  [744] = {x=191.932, y=87.653, z=110, rx=-180, rz=-113.182, shoulder=lefty, elbow=epositive, wrist=wpositive, fatherId=fReference[0]}
  [745] = {x=195.886, y=78.421, z=110, rx=-180, rz=-110.455, shoulder=lefty, elbow=epositive, wrist=wpositive, fatherId=fReference[0]}
  [746] = {x=199.395, y=69.011, z=110, rx=-180, rz=-107.727, shoulder=lefty, elbow=epositive, wrist=wpositive, fatherId=fReference[0]}
  [747] = {x=202.453, y=59.446, z=110, rx=-180, rz=-105, shoulder=lefty, elbow=epositive, wrist=wpositive, fatherId=fReference[0]}
  [748] = {x=205.052, y=49.745, z=110, rx=-180, rz=-102.273, shoulder=lefty, elbow=epositive, wrist=wpositive, fatherId=fReference[0]}
  [749] = {x=207.187, y=39.932, z=110, rx=-180, rz=-99.545, shoulder=lefty, elbow=epositive, wrist=wpositive, fatherId=fReference[0]}
  [750] = {x=208.852, y=30.028, z=110, rx=-180, rz=-96.818, shoulder=lefty, elbow=epositive, wrist=wpositive, fatherId=fReference[0]}
  [751] = {x=210.045, y=20.057, z=110, rx=-180, rz=-94.091, shoulder=lefty, elbow=epositive, wrist=wpositive, fatherId=fReference[0]}
  [752] = {x=210.761, y=10.04, z=110, rx=-180, rz=-91.364, shoulder=lefty, elbow=epositive, wrist=wpositive, fatherId=fReference[0]}
  [753] = {x=211, z=110, rx=180, rz=-88.636, shoulder=lefty, elbow=epositive, wrist=wpositive, fatherId=fReference[0]}
  [754] = {x=210.761, y=-10.04, z=110, rx=180, rz=-85.909, shoulder=lefty, elbow=epositive, wrist=wpositive, fatherId=fReference[0]}
  [755] = {x=210.045, y=-20.057, z=110, rx=180, rz=-83.182, shoulder=lefty, elbow=epositive, wrist=wpositive, fatherId=fReference[0]}
  [756] = {x=208.852, y=-30.028, z=110, rx=180, rz=-80.455, shoulder=lefty, elbow=epositive, wrist=wpositive, fatherId=fReference[0]}
  [757] = {x=207.187, y=-39.932, z=110, rx=180, rz=-77.727, shoulder=lefty, elbow=epositive, wrist=wpositive, fatherId=fReference[0]}
  [758] = {x=205.052, y=-49.745, z=110, rx=180, rz=-75, shoulder=lefty, elbow=epositive, wrist=wpositive, fatherId=fReference[0]}
  [759] = {x=202.453, y=-59.446, z=110, rx=180, rz=-72.273, shoulder=lefty, elbow=epositive, wrist=wpositive, fatherId=fReference[0]}
  [760] = {x=199.395, y=-69.011, z=110, rx=180, rz=-69.545, shoulder=lefty, elbow=epositive, wrist=wpositive, fatherId=fReference[0]}
  [761] = {x=195.886, y=-78.421, z=110, rx=180, rz=-66.818, shoulder=lefty, elbow=epositive, wrist=wpositive, fatherId=fReference[0]}
  [762] = {x=191.932, y=-87.653, z=110, rx=180, rz=-64.091, shoulder=lefty, elbow=epositive, wrist=wpositive, fatherId=fReference[0]}
  [763] = {x=187.544, y=-96.686, z=110, rx=180, rz=-61.364, shoulder=lefty, elbow=epositive, wrist=wpositive, fatherId=fReference[0]}
  [764] = {x=182.731, y=-105.5, z=110, rx=-180, rz=-58.636, shoulder=lefty, elbow=epositive, wrist=wpositive, fatherId=fReference[0]}
  [765] = {x=177.505, y=-114.075, z=110, rx=180, rz=-55.909, shoulder=lefty, elbow=epositive, wrist=wpositive, fatherId=fReference[0]}
  [766] = {x=171.876, y=-122.392, z=110, rx=180, rz=-53.182, shoulder=lefty, elbow=epositive, wrist=wpositive, fatherId=fReference[0]}
  [767] = {x=165.857, y=-130.432, z=110, rx=180, rz=-50.455, shoulder=lefty, elbow=epositive, wrist=wpositive, fatherId=fReference[0]}
  [768] = {x=159.463, y=-138.176, z=110, rx=180, rz=-47.727, shoulder=lefty, elbow=epositive, wrist=wpositive, fatherId=fReference[0]}
  [769] = {x=152.708, y=-145.607, z=110, rx=180, rz=-45, shoulder=lefty, elbow=epositive, wrist=wpositive, fatherId=fReference[0]}
  [770] = {x=145.607, y=-152.708, z=110, rx=180, rz=-42.273, shoulder=lefty, elbow=epositive, wrist=wpositive, fatherId=fReference[0]}
  [771] = {x=138.176, y=-159.463, z=110, rx=180, rz=-39.545, shoulder=lefty, elbow=epositive, wrist=wpositive, fatherId=fReference[0]}
  [772] = {x=130.432, y=-165.857, z=110, rx=-180, rz=-36.818, shoulder=lefty, elbow=epositive, wrist=wpositive, fatherId=fReference[0]}
  [773] = {x=122.392, y=-171.876, z=110, rx=180, rz=-34.091, shoulder=lefty, elbow=epositive, wrist=wpositive, fatherId=fReference[0]}
  [774] = {x=114.075, y=-177.505, z=110, rx=180, rz=-31.364, shoulder=lefty, elbow=epositive, wrist=wpositive, fatherId=fReference[0]}
  [775] = {x=105.5, y=-182.731, z=110, rx=-180, rz=-28.636, shoulder=lefty, elbow=epositive, wrist=wpositive, fatherId=fReference[0]}
  [776] = {x=96.686, y=-187.544, z=110, rx=-180, rz=-25.909, shoulder=lefty, elbow=epositive, wrist=wpositive, fatherId=fReference[0]}
  [777] = {x=87.653, y=-191.932, z=110, rx=180, rz=-23.182, shoulder=lefty, elbow=epositive, wrist=wpositive, fatherId=fReference[0]}
  [778] = {x=78.421, y=-195.886, z=110, rx=180, rz=-20.455, shoulder=lefty, elbow=epositive, wrist=wpositive, fatherId=fReference[0]}
  [779] = {x=69.011, y=-199.395, z=110, rx=-180, rz=-17.727, shoulder=lefty, elbow=epositive, wrist=wpositive, fatherId=fReference[0]}
  [780] = {x=59.446, y=-202.453, z=110, rx=180, rz=-15, shoulder=lefty, elbow=epositive, wrist=wpositive, fatherId=fReference[0]}
  [781] = {x=49.745, y=-205.052, z=110, rx=-180, rz=-12.273, shoulder=lefty, elbow=epositive, wrist=wpositive, fatherId=fReference[0]}
  [782] = {x=39.932, y=-207.187, z=110, rx=180, rz=-9.545, shoulder=lefty, elbow=epositive, wrist=wpositive, fatherId=fReference[0]}
  [783] = {x=30.028, y=-208.852, z=110, rx=-180, rz=-6.818, shoulder=lefty, elbow=epositive, wrist=wpositive, fatherId=fReference[0]}
  [784] = {x=20.057, y=-210.045, z=110, rx=180, rz=-4.091, shoulder=lefty, elbow=epositive, wrist=wpositive, fatherId=fReference[0]}
  [785] = {x=10.04, y=-210.761, z=110, rx=180, rz=-1.364, shoulder=lefty, elbow=epositive, wrist=wpositive, fatherId=fReference[0]}
  [786] = {y=-211, z=110, rx=-180, rz=1.364, shoulder=lefty, elbow=epositive, wrist=wpositive, fatherId=fReference[0]}
  [787] = {x=-10.04, y=-210.761, z=110, rx=-180, rz=4.091, shoulder=lefty, elbow=epositive, wrist=wpositive, fatherId=fReference[0]}
  [788] = {x=-20.057, y=-210.045, z=110, rx=-180, rz=6.818, shoulder=lefty, elbow=epositive, wrist=wpositive, fatherId=fReference[0]}
  [789] = {x=-30.028, y=-208.852, z=110, rx=-180, rz=9.545, shoulder=lefty, elbow=epositive, wrist=wpositive, fatherId=fReference[0]}
  [790] = {x=-39.932, y=-207.187, z=110, rx=-180, rz=12.273, shoulder=lefty, elbow=epositive, wrist=wpositive, fatherId=fReference[0]}
  [791] = {x=-49.745, y=-205.052, z=110, rx=-180, rz=15, shoulder=lefty, elbow=epositive, wrist=wpositive, fatherId=fReference[0]}
  [792] = {x=-59.446, y=-202.453, z=110, rx=-180, rz=17.727, shoulder=lefty, elbow=epositive, wrist=wpositive, fatherId=fReference[0]}
  [793] = {x=-69.011, y=-199.395, z=110, rx=-180, rz=20.455, shoulder=lefty, elbow=epositive, wrist=wpositive, fatherId=fReference[0]}
  [794] = {x=-78.421, y=-195.886, z=110, rx=-180, rz=23.182, shoulder=lefty, elbow=epositive, wrist=wpositive, fatherId=fReference[0]}
  [795] = {x=-87.653, y=-191.932, z=110, rx=-180, rz=25.909, shoulder=lefty, elbow=epositive, wrist=wpositive, fatherId=fReference[0]}
  [796] = {x=-96.686, y=-187.544, z=110, rx=-180, rz=28.636, shoulder=lefty, elbow=epositive, wrist=wpositive, fatherId=fReference[0]}
  [797] = {x=-105.5, y=-182.731, z=110, rx=-180, rz=31.364, shoulder=lefty, elbow=epositive, wrist=wpositive, fatherId=fReference[0]}
  [798] = {x=-114.075, y=-177.505, z=110, rx=-180, rz=34.091, shoulder=lefty, elbow=epositive, wrist=wpositive, fatherId=fReference[0]}
  [799] = {x=-122.392, y=-171.876, z=110, rx=-180, rz=36.818, shoulder=lefty, elbow=epositive, wrist=wpositive, fatherId=fReference[0]}
  [800] = {x=-130.432, y=-165.857, z=110, rx=-180, rz=39.545, shoulder=lefty, elbow=epositive, wrist=wpositive, fatherId=fReference[0]}
  [801] = {x=-138.176, y=-159.463, z=110, rx=-180, rz=42.273, shoulder=lefty, elbow=epositive, wrist=wpositive, fatherId=fReference[0]}
  [802] = {x=-145.607, y=-152.708, z=110, rx=-180, rz=45, shoulder=lefty, elbow=epositive, wrist=wpositive, fatherId=fReference[0]}
  [803] = {x=-152.708, y=-145.607, z=110, rx=-180, rz=47.727, shoulder=lefty, elbow=epositive, wrist=wpositive, fatherId=fReference[0]}
  [804] = {x=-159.463, y=-138.176, z=110, rx=180, rz=50.455, shoulder=lefty, elbow=epositive, wrist=wpositive, fatherId=fReference[0]}
  [805] = {x=-165.857, y=-130.432, z=110, rx=-180, rz=53.182, shoulder=lefty, elbow=epositive, wrist=wpositive, fatherId=fReference[0]}
  [806] = {x=-171.876, y=-122.392, z=110, rx=-180, rz=55.909, shoulder=lefty, elbow=epositive, wrist=wpositive, fatherId=fReference[0]}
  [807] = {x=-177.505, y=-114.075, z=110, rx=-180, rz=58.636, shoulder=lefty, elbow=epositive, wrist=wpositive, fatherId=fReference[0]}
  [808] = {x=-182.731, y=-105.5, z=110, rx=-180, rz=61.364, shoulder=lefty, elbow=epositive, wrist=wpositive, fatherId=fReference[0]}
  [809] = {x=-187.544, y=-96.686, z=110, rx=-180, rz=64.091, shoulder=lefty, elbow=epositive, wrist=wpositive, fatherId=fReference[0]}
  [810] = {x=-191.932, y=-87.653, z=110, rx=180, rz=66.818, shoulder=lefty, elbow=epositive, wrist=wpositive, fatherId=fReference[0]}
  [811] = {x=-195.886, y=-78.421, z=110, rx=-180, rz=69.545, shoulder=lefty, elbow=epositive, wrist=wpositive, fatherId=fReference[0]}
  [812] = {x=-199.395, y=-69.011, z=110, rx=-180, rz=72.273, shoulder=lefty, elbow=epositive, wrist=wpositive, fatherId=fReference[0]}
  [813] = {x=-202.453, y=-59.446, z=110, rx=-180, rz=75, shoulder=lefty, elbow=epositive, wrist=wpositive, fatherId=fReference[0]}
  [814] = {x=-205.052, y=-49.745, z=110, rx=-180, rz=77.727, shoulder=lefty, elbow=epositive, wrist=wpositive, fatherId=fReference[0]}
  [815] = {x=-207.187, y=-39.932, z=110, rx=-180, rz=80.455, shoulder=lefty, elbow=epositive, wrist=wpositive, fatherId=fReference[0]}
  [816] = {x=-208.852, y=-30.028, z=110, rx=-180, rz=83.182, shoulder=lefty, elbow=epositive, wrist=wpositive, fatherId=fReference[0]}
  [817] = {x=-210.045, y=-20.057, z=110, rx=-180, rz=85.909, shoulder=lefty, elbow=epositive, wrist=wpositive, fatherId=fReference[0]}
  [818] = {x=-210.761, y=-10.04, z=110, rx=-180, rz=88.636, shoulder=lefty, elbow=epositive, wrist=wpositive, fatherId=fReference[0]}
  [819] = {x=-211, z=110, rx=-180, rz=88.636, shoulder=lefty, elbow=epositive, wrist=wpositive, fatherId=fReference[0]}
  [820] = {x=-211, z=110, rx=-180, rz=88.636, shoulder=lefty, elbow=epositive, wrist=wpositive, fatherId=fReference[0]}
  [821] = {x=-211, z=210, rx=-180, rz=88.636, shoulder=lefty, elbow=epositive, wrist=wpositive, fatherId=fReference[0]}
  [822] = {x=-211, z=232, rx=-180, rz=88.636, shoulder=lefty, elbow=epositive, wrist=wpositive, fatherId=fReference[0]}
  [823] = {x=-211, z=132, rx=-180, rz=88.636, shoulder=lefty, elbow=epositive, wrist=wpositive, fatherId=fReference[0]}
  [824] = {x=-211, z=132, rx=-180, rz=88.636, shoulder=lefty, elbow=epositive, wrist=wpositive, fatherId=fReference[0]}
  [825] = {x=-210.761, y=-10.04, z=132, rx=-180, rz=85.909, shoulder=lefty, elbow=epositive, wrist=wpositive, fatherId=fReference[0]}
  [826] = {x=-210.045, y=-20.057, z=132, rx=-180, rz=83.182, shoulder=lefty, elbow=epositive, wrist=wpositive, fatherId=fReference[0]}
  [827] = {x=-208.852, y=-30.028, z=132, rx=-180, rz=80.455, shoulder=lefty, elbow=epositive, wrist=wpositive, fatherId=fReference[0]}
  [828] = {x=-207.187, y=-39.932, z=132, rx=-180, rz=77.727, shoulder=lefty, elbow=epositive, wrist=wpositive, fatherId=fReference[0]}
  [829] = {x=-205.052, y=-49.745, z=132, rx=-180, rz=75, shoulder=lefty, elbow=epositive, wrist=wpositive, fatherId=fReference[0]}
  [830] = {x=-202.453, y=-59.446, z=132, rx=-180, rz=72.273, shoulder=lefty, elbow=epositive, wrist=wpositive, fatherId=fReference[0]}
  [831] = {x=-199.395, y=-69.011, z=132, rx=-180, rz=69.545, shoulder=lefty, elbow=epositive, wrist=wpositive, fatherId=fReference[0]}
  [832] = {x=-195.886, y=-78.421, z=132, rx=-180, rz=66.818, shoulder=lefty, elbow=epositive, wrist=wpositive, fatherId=fReference[0]}
  [833] = {x=-191.932, y=-87.653, z=132, rx=180, rz=64.091, shoulder=lefty, elbow=epositive, wrist=wpositive, fatherId=fReference[0]}
  [834] = {x=-187.544, y=-96.686, z=132, rx=-180, rz=61.364, shoulder=lefty, elbow=epositive, wrist=wpositive, fatherId=fReference[0]}
  [835] = {x=-182.731, y=-105.5, z=132, rx=-180, rz=58.636, shoulder=lefty, elbow=epositive, wrist=wpositive, fatherId=fReference[0]}
  [836] = {x=-177.505, y=-114.075, z=132, rx=180, rz=55.909, shoulder=lefty, elbow=epositive, wrist=wpositive, fatherId=fReference[0]}
  [837] = {x=-171.876, y=-122.392, z=132, rx=-180, rz=53.182, shoulder=lefty, elbow=epositive, wrist=wpositive, fatherId=fReference[0]}
  [838] = {x=-165.857, y=-130.432, z=132, rx=-180, rz=50.455, shoulder=lefty, elbow=epositive, wrist=wpositive, fatherId=fReference[0]}
  [839] = {x=-159.463, y=-138.176, z=132, rx=-180, rz=47.727, shoulder=lefty, elbow=epositive, wrist=wpositive, fatherId=fReference[0]}
  [840] = {x=-152.708, y=-145.607, z=132, rx=-180, rz=45, shoulder=lefty, elbow=epositive, wrist=wpositive, fatherId=fReference[0]}
  [841] = {x=-145.607, y=-152.708, z=132, rx=-180, rz=42.273, shoulder=lefty, elbow=epositive, wrist=wpositive, fatherId=fReference[0]}
  [842] = {x=-138.176, y=-159.463, z=132, rx=180, rz=39.545, shoulder=lefty, elbow=epositive, wrist=wpositive, fatherId=fReference[0]}
  [843] = {x=-130.432, y=-165.857, z=132, rx=-180, rz=36.818, shoulder=lefty, elbow=epositive, wrist=wpositive, fatherId=fReference[0]}
  [844] = {x=-122.392, y=-171.876, z=132, rx=-180, rz=34.091, shoulder=lefty, elbow=epositive, wrist=wpositive, fatherId=fReference[0]}
  [845] = {x=-114.075, y=-177.505, z=132, rx=-180, rz=31.364, shoulder=lefty, elbow=epositive, wrist=wpositive, fatherId=fReference[0]}
  [846] = {x=-105.5, y=-182.731, z=132, rx=180, rz=28.636, shoulder=lefty, elbow=epositive, wrist=wpositive, fatherId=fReference[0]}
  [847] = {x=-96.686, y=-187.544, z=132, rx=-180, rz=25.909, shoulder=lefty, elbow=epositive, wrist=wpositive, fatherId=fReference[0]}
  [848] = {x=-87.653, y=-191.932, z=132, rx=180, rz=23.182, shoulder=lefty, elbow=epositive, wrist=wpositive, fatherId=fReference[0]}
  [849] = {x=-78.421, y=-195.886, z=132, rx=180, rz=20.455, shoulder=lefty, elbow=epositive, wrist=wpositive, fatherId=fReference[0]}
  [850] = {x=-69.011, y=-199.395, z=132, rx=-180, rz=17.727, shoulder=lefty, elbow=epositive, wrist=wpositive, fatherId=fReference[0]}
  [851] = {x=-59.446, y=-202.453, z=132, rx=180, rz=15, shoulder=lefty, elbow=epositive, wrist=wpositive, fatherId=fReference[0]}
  [852] = {x=-49.745, y=-205.052, z=132, rx=-180, rz=12.273, shoulder=lefty, elbow=epositive, wrist=wpositive, fatherId=fReference[0]}
  [853] = {x=-39.932, y=-207.187, z=132, rx=180, rz=9.545, shoulder=lefty, elbow=epositive, wrist=wpositive, fatherId=fReference[0]}
  [854] = {x=-30.028, y=-208.852, z=132, rx=-180, rz=6.818, shoulder=lefty, elbow=epositive, wrist=wpositive, fatherId=fReference[0]}
  [855] = {x=-20.057, y=-210.045, z=132, rx=180, rz=4.091, shoulder=lefty, elbow=epositive, wrist=wpositive, fatherId=fReference[0]}
  [856] = {x=-10.04, y=-210.761, z=132, rx=-180, rz=1.364, shoulder=lefty, elbow=epositive, wrist=wpositive, fatherId=fReference[0]}
  [857] = {y=-211, z=132, rx=180, rz=-1.364, shoulder=lefty, elbow=epositive, wrist=wpositive, fatherId=fReference[0]}
  [858] = {x=10.04, y=-210.761, z=132, rx=180, rz=-4.091, shoulder=lefty, elbow=epositive, wrist=wpositive, fatherId=fReference[0]}
  [859] = {x=20.057, y=-210.045, z=132, rx=180, rz=-6.818, shoulder=lefty, elbow=epositive, wrist=wpositive, fatherId=fReference[0]}
  [860] = {x=30.028, y=-208.852, z=132, rx=180, rz=-9.545, shoulder=lefty, elbow=epositive, wrist=wpositive, fatherId=fReference[0]}
  [861] = {x=39.932, y=-207.187, z=132, rx=180, rz=-12.273, shoulder=lefty, elbow=epositive, wrist=wpositive, fatherId=fReference[0]}
  [862] = {x=49.745, y=-205.052, z=132, rx=-180, rz=-15, shoulder=lefty, elbow=epositive, wrist=wpositive, fatherId=fReference[0]}
  [863] = {x=59.446, y=-202.453, z=132, rx=-180, rz=-17.727, shoulder=lefty, elbow=epositive, wrist=wpositive, fatherId=fReference[0]}
  [864] = {x=69.011, y=-199.395, z=132, rx=180, rz=-20.455, shoulder=lefty, elbow=epositive, wrist=wpositive, fatherId=fReference[0]}
  [865] = {x=78.421, y=-195.886, z=132, rx=-180, rz=-23.182, shoulder=lefty, elbow=epositive, wrist=wpositive, fatherId=fReference[0]}
  [866] = {x=87.653, y=-191.932, z=132, rx=-180, rz=-25.909, shoulder=lefty, elbow=epositive, wrist=wpositive, fatherId=fReference[0]}
  [867] = {x=96.686, y=-187.544, z=132, rx=-180, rz=-28.636, shoulder=lefty, elbow=epositive, wrist=wpositive, fatherId=fReference[0]}
  [868] = {x=105.5, y=-182.731, z=132, rx=180, rz=-31.364, shoulder=lefty, elbow=epositive, wrist=wpositive, fatherId=fReference[0]}
  [869] = {x=114.075, y=-177.505, z=132, rx=180, rz=-34.091, shoulder=lefty, elbow=epositive, wrist=wpositive, fatherId=fReference[0]}
  [870] = {x=122.392, y=-171.876, z=132, rx=180, rz=-36.818, shoulder=lefty, elbow=epositive, wrist=wpositive, fatherId=fReference[0]}
  [871] = {x=130.432, y=-165.857, z=132, rx=180, rz=-39.545, shoulder=lefty, elbow=epositive, wrist=wpositive, fatherId=fReference[0]}
  [872] = {x=138.176, y=-159.463, z=132, rx=180, rz=-42.273, shoulder=lefty, elbow=epositive, wrist=wpositive, fatherId=fReference[0]}
  [873] = {x=145.607, y=-152.708, z=132, rx=180, rz=-45, shoulder=lefty, elbow=epositive, wrist=wpositive, fatherId=fReference[0]}
  [874] = {x=152.708, y=-145.607, z=132, rx=180, rz=-47.727, shoulder=lefty, elbow=epositive, wrist=wpositive, fatherId=fReference[0]}
  [875] = {x=159.463, y=-138.176, z=132, rx=180, rz=-50.455, shoulder=lefty, elbow=epositive, wrist=wpositive, fatherId=fReference[0]}
  [876] = {x=165.857, y=-130.432, z=132, rx=180, rz=-53.182, shoulder=lefty, elbow=epositive, wrist=wpositive, fatherId=fReference[0]}
  [877] = {x=171.876, y=-122.392, z=132, rx=180, rz=-55.909, shoulder=lefty, elbow=epositive, wrist=wpositive, fatherId=fReference[0]}
  [878] = {x=177.505, y=-114.075, z=132, rx=180, rz=-58.636, shoulder=lefty, elbow=epositive, wrist=wpositive, fatherId=fReference[0]}
  [879] = {x=182.731, y=-105.5, z=132, rx=180, rz=-61.364, shoulder=lefty, elbow=epositive, wrist=wpositive, fatherId=fReference[0]}
  [880] = {x=187.544, y=-96.686, z=132, rx=180, rz=-64.091, shoulder=lefty, elbow=epositive, wrist=wpositive, fatherId=fReference[0]}
  [881] = {x=191.932, y=-87.653, z=132, rx=-180, rz=-66.818, shoulder=lefty, elbow=epositive, wrist=wpositive, fatherId=fReference[0]}
  [882] = {x=195.886, y=-78.421, z=132, rx=180, rz=-69.545, shoulder=lefty, elbow=epositive, wrist=wpositive, fatherId=fReference[0]}
  [883] = {x=199.395, y=-69.011, z=132, rx=180, rz=-72.273, shoulder=lefty, elbow=epositive, wrist=wpositive, fatherId=fReference[0]}
  [884] = {x=202.453, y=-59.446, z=132, rx=180, rz=-75, shoulder=lefty, elbow=epositive, wrist=wpositive, fatherId=fReference[0]}
  [885] = {x=205.052, y=-49.745, z=132, rx=180, rz=-77.727, shoulder=lefty, elbow=epositive, wrist=wpositive, fatherId=fReference[0]}
  [886] = {x=207.187, y=-39.932, z=132, rx=180, rz=-80.455, shoulder=lefty, elbow=epositive, wrist=wpositive, fatherId=fReference[0]}
  [887] = {x=208.852, y=-30.028, z=132, rx=180, rz=-83.182, shoulder=lefty, elbow=epositive, wrist=wpositive, fatherId=fReference[0]}
  [888] = {x=210.045, y=-20.057, z=132, rx=180, rz=-85.909, shoulder=lefty, elbow=epositive, wrist=wpositive, fatherId=fReference[0]}
  [889] = {x=210.761, y=-10.04, z=132, rx=180, rz=-88.636, shoulder=lefty, elbow=epositive, wrist=wpositive, fatherId=fReference[0]}
  [890] = {x=211, z=132, rx=-180, rz=-91.364, shoulder=lefty, elbow=epositive, wrist=wpositive, fatherId=fReference[0]}
  [891] = {x=210.761, y=10.04, z=132, rx=-180, rz=-94.091, shoulder=lefty, elbow=epositive, wrist=wpositive, fatherId=fReference[0]}
  [892] = {x=210.045, y=20.057, z=132, rx=-180, rz=-96.818, shoulder=lefty, elbow=epositive, wrist=wpositive, fatherId=fReference[0]}
  [893] = {x=208.852, y=30.028, z=132, rx=-180, rz=-99.545, shoulder=lefty, elbow=epositive, wrist=wpositive, fatherId=fReference[0]}
  [894] = {x=207.187, y=39.932, z=132, rx=-180, rz=-102.273, shoulder=lefty, elbow=epositive, wrist=wpositive, fatherId=fReference[0]}
  [895] = {x=205.052, y=49.745, z=132, rx=-180, rz=-105, shoulder=lefty, elbow=epositive, wrist=wpositive, fatherId=fReference[0]}
  [896] = {x=202.453, y=59.446, z=132, rx=-180, rz=-107.727, shoulder=lefty, elbow=epositive, wrist=wpositive, fatherId=fReference[0]}
  [897] = {x=199.395, y=69.011, z=132, rx=-180, rz=-110.455, shoulder=lefty, elbow=epositive, wrist=wpositive, fatherId=fReference[0]}
  [898] = {x=195.886, y=78.421, z=132, rx=-180, rz=-113.182, shoulder=lefty, elbow=epositive, wrist=wpositive, fatherId=fReference[0]}
  [899] = {x=191.932, y=87.653, z=132, rx=-180, rz=-115.909, shoulder=lefty, elbow=epositive, wrist=wpositive, fatherId=fReference[0]}
  [900] = {x=187.544, y=96.686, z=132, rx=-180, rz=-118.636, shoulder=lefty, elbow=epositive, wrist=wpositive, fatherId=fReference[0]}
  [901] = {x=182.731, y=105.5, z=132, rx=-180, rz=-121.364, shoulder=lefty, elbow=epositive, wrist=wpositive, fatherId=fReference[0]}
  [902] = {x=177.505, y=114.075, z=132, rx=-180, rz=-124.091, shoulder=lefty, elbow=epositive, wrist=wpositive, fatherId=fReference[0]}
  [903] = {x=171.876, y=122.392, z=132, rx=-180, rz=-126.818, shoulder=lefty, elbow=epositive, wrist=wpositive, fatherId=fReference[0]}
  [904] = {x=165.857, y=130.432, z=132, rx=-180, rz=-129.545, shoulder=lefty, elbow=epositive, wrist=wpositive, fatherId=fReference[0]}
  [905] = {x=159.463, y=138.176, z=132, rx=-180, rz=-132.273, shoulder=lefty, elbow=epositive, wrist=wpositive, fatherId=fReference[0]}
  [906] = {x=152.708, y=145.607, z=132, rx=-180, rz=-135, shoulder=lefty, elbow=epositive, wrist=wpositive, fatherId=fReference[0]}
  [907] = {x=145.607, y=152.708, z=132, rx=-180, rz=-137.727, shoulder=lefty, elbow=epositive, wrist=wpositive, fatherId=fReference[0]}
  [908] = {x=138.176, y=159.463, z=132, rx=-180, rz=-140.455, shoulder=lefty, elbow=epositive, wrist=wpositive, fatherId=fReference[0]}
  [909] = {x=130.432, y=165.857, z=132, rx=180, rz=-143.182, shoulder=lefty, elbow=epositive, wrist=wpositive, fatherId=fReference[0]}
  [910] = {x=122.392, y=171.876, z=132, rx=-180, rz=-145.909, shoulder=lefty, elbow=epositive, wrist=wpositive, fatherId=fReference[0]}
  [911] = {x=114.075, y=177.505, z=132, rx=180, rz=-148.636, shoulder=lefty, elbow=epositive, wrist=wpositive, fatherId=fReference[0]}
  [912] = {x=105.5, y=182.731, z=132, rx=180, rz=-151.364, shoulder=lefty, elbow=epositive, wrist=wpositive, fatherId=fReference[0]}
  [913] = {x=96.686, y=187.544, z=132, rx=-180, rz=-154.091, shoulder=lefty, elbow=epositive, wrist=wpositive, fatherId=fReference[0]}
  [914] = {x=87.653, y=191.932, z=132, rx=-180, rz=-156.818, shoulder=lefty, elbow=epositive, wrist=wpositive, fatherId=fReference[0]}
  [915] = {x=78.421, y=195.886, z=132, rx=-180, rz=-159.545, shoulder=lefty, elbow=epositive, wrist=wpositive, fatherId=fReference[0]}
  [916] = {x=69.011, y=199.395, z=132, rx=-180, rz=-162.273, shoulder=lefty, elbow=epositive, wrist=wpositive, fatherId=fReference[0]}
  [917] = {x=59.446, y=202.453, z=132, rx=-180, rz=-165, shoulder=lefty, elbow=epositive, wrist=wpositive, fatherId=fReference[0]}
  [918] = {x=49.745, y=205.052, z=132, rx=180, rz=-167.727, shoulder=lefty, elbow=epositive, wrist=wpositive, fatherId=fReference[0]}
  [919] = {x=39.932, y=207.187, z=132, rx=180, rz=-170.455, shoulder=lefty, elbow=epositive, wrist=wpositive, fatherId=fReference[0]}
  [920] = {x=30.028, y=208.852, z=132, rx=-180, rz=-173.182, shoulder=lefty, elbow=epositive, wrist=wpositive, fatherId=fReference[0]}
  [921] = {x=20.057, y=210.045, z=132, rx=-180, rz=-175.909, shoulder=lefty, elbow=epositive, wrist=wpositive, fatherId=fReference[0]}
  [922] = {x=10.04, y=210.761, z=132, rx=-180, rz=-178.636, shoulder=lefty, elbow=epositive, wrist=wpositive, fatherId=fReference[0]}
  [923] = {y=211, z=132, rx=-180, rz=178.636, shoulder=lefty, elbow=epositive, wrist=wpositive, fatherId=fReference[0]}
  [924] = {x=-10.04, y=210.761, z=132, rx=180, rz=175.909, shoulder=lefty, elbow=epositive, wrist=wpositive, fatherId=fReference[0]}
  [925] = {x=-20.057, y=210.045, z=132, rx=180, rz=173.182, shoulder=lefty, elbow=epositive, wrist=wpositive, fatherId=fReference[0]}
  [926] = {x=-30.028, y=208.852, z=132, rx=180, rz=170.455, shoulder=lefty, elbow=epositive, wrist=wpositive, fatherId=fReference[0]}
  [927] = {x=-39.932, y=207.187, z=132, rx=180, rz=167.727, shoulder=lefty, elbow=epositive, wrist=wpositive, fatherId=fReference[0]}
  [928] = {x=-49.745, y=205.052, z=132, rx=-180, rz=165, shoulder=lefty, elbow=epositive, wrist=wpositive, fatherId=fReference[0]}
  [929] = {x=-59.446, y=202.453, z=132, rx=180, rz=162.273, shoulder=lefty, elbow=epositive, wrist=wpositive, fatherId=fReference[0]}
  [930] = {x=-69.011, y=199.395, z=132, rx=180, rz=159.545, shoulder=lefty, elbow=epositive, wrist=wpositive, fatherId=fReference[0]}
  [931] = {x=-78.421, y=195.886, z=132, rx=-180, rz=156.818, shoulder=lefty, elbow=epositive, wrist=wpositive, fatherId=fReference[0]}
  [932] = {x=-87.653, y=191.932, z=132, rx=180, rz=154.091, shoulder=lefty, elbow=epositive, wrist=wpositive, fatherId=fReference[0]}
  [933] = {x=-96.686, y=187.544, z=132, rx=-180, rz=151.364, shoulder=lefty, elbow=epositive, wrist=wpositive, fatherId=fReference[0]}
  [934] = {x=-105.5, y=182.731, z=132, rx=180, rz=148.636, shoulder=lefty, elbow=epositive, wrist=wpositive, fatherId=fReference[0]}
  [935] = {x=-114.075, y=177.505, z=132, rx=-180, rz=145.909, shoulder=lefty, elbow=epositive, wrist=wpositive, fatherId=fReference[0]}
  [936] = {x=-122.392, y=171.876, z=132, rx=-180, rz=143.182, shoulder=lefty, elbow=epositive, wrist=wpositive, fatherId=fReference[0]}
  [937] = {x=-130.432, y=165.857, z=132, rx=-180, rz=140.455, shoulder=lefty, elbow=epositive, wrist=wpositive, fatherId=fReference[0]}
  [938] = {x=-138.176, y=159.463, z=132, rx=180, rz=137.727, shoulder=lefty, elbow=epositive, wrist=wpositive, fatherId=fReference[0]}
  [939] = {x=-145.607, y=152.708, z=132, rx=180, rz=135, shoulder=lefty, elbow=epositive, wrist=wpositive, fatherId=fReference[0]}
  [940] = {x=-152.708, y=145.607, z=132, rx=180, rz=132.273, shoulder=lefty, elbow=epositive, wrist=wpositive, fatherId=fReference[0]}
  [941] = {x=-159.463, y=138.176, z=132, rx=180, rz=129.545, shoulder=lefty, elbow=epositive, wrist=wpositive, fatherId=fReference[0]}
  [942] = {x=-165.857, y=130.432, z=132, rx=180, rz=126.818, shoulder=lefty, elbow=epositive, wrist=wpositive, fatherId=fReference[0]}
  [943] = {x=-171.876, y=122.392, z=132, rx=180, rz=124.091, shoulder=lefty, elbow=epositive, wrist=wpositive, fatherId=fReference[0]}
  [944] = {x=-177.505, y=114.075, z=132, rx=180, rz=121.364, shoulder=lefty, elbow=epositive, wrist=wpositive, fatherId=fReference[0]}
  [945] = {x=-182.731, y=105.5, z=132, rx=180, rz=118.636, shoulder=lefty, elbow=epositive, wrist=wpositive, fatherId=fReference[0]}
  [946] = {x=-187.544, y=96.686, z=132, rx=180, rz=115.909, shoulder=lefty, elbow=epositive, wrist=wpositive, fatherId=fReference[0]}
  [947] = {x=-191.932, y=87.653, z=132, rx=180, rz=113.182, shoulder=lefty, elbow=epositive, wrist=wpositive, fatherId=fReference[0]}
  [948] = {x=-195.886, y=78.421, z=132, rx=180, rz=110.455, shoulder=lefty, elbow=epositive, wrist=wpositive, fatherId=fReference[0]}
  [949] = {x=-199.395, y=69.011, z=132, rx=180, rz=107.727, shoulder=lefty, elbow=epositive, wrist=wpositive, fatherId=fReference[0]}
  [950] = {x=-202.453, y=59.446, z=132, rx=180, rz=105, shoulder=lefty, elbow=epositive, wrist=wpositive, fatherId=fReference[0]}
  [951] = {x=-205.052, y=49.745, z=132, rx=180, rz=102.273, shoulder=lefty, elbow=epositive, wrist=wpositive, fatherId=fReference[0]}
  [952] = {x=-207.187, y=39.932, z=132, rx=180, rz=99.545, shoulder=lefty, elbow=epositive, wrist=wpositive, fatherId=fReference[0]}
  [953] = {x=-208.852, y=30.028, z=132, rx=180, rz=96.818, shoulder=lefty, elbow=epositive, wrist=wpositive, fatherId=fReference[0]}
  [954] = {x=-210.045, y=20.057, z=132, rx=180, rz=94.091, shoulder=lefty, elbow=epositive, wrist=wpositive, fatherId=fReference[0]}
  [955] = {x=-210.761, y=10.04, z=132, rx=180, rz=91.364, shoulder=lefty, elbow=epositive, wrist=wpositive, fatherId=fReference[0]}
  [956] = {x=-211, z=132, rx=180, rz=91.364, shoulder=lefty, elbow=epositive, wrist=wpositive, fatherId=fReference[0]}
  [957] = {x=-211, z=132, rx=180, rz=91.364, shoulder=lefty, elbow=epositive, wrist=wpositive, fatherId=fReference[0]}
  [958] = {x=-211, z=232, rx=180, rz=91.364, shoulder=lefty, elbow=epositive, wrist=wpositive, fatherId=fReference[0]}
  [959] = {x=-211, z=254, rx=180, rz=91.364, shoulder=lefty, elbow=epositive, wrist=wpositive, fatherId=fReference[0]}
  [960] = {x=-211, z=154, rx=180, rz=91.364, shoulder=lefty, elbow=epositive, wrist=wpositive, fatherId=fReference[0]}
  [961] = {x=-211, z=154, rx=180, rz=91.364, shoulder=lefty, elbow=epositive, wrist=wpositive, fatherId=fReference[0]}
  [962] = {x=-210.761, y=10.04, z=154, rx=180, rz=94.091, shoulder=lefty, elbow=epositive, wrist=wpositive, fatherId=fReference[0]}
  [963] = {x=-210.045, y=20.057, z=154, rx=180, rz=96.818, shoulder=lefty, elbow=epositive, wrist=wpositive, fatherId=fReference[0]}
  [964] = {x=-208.852, y=30.028, z=154, rx=180, rz=99.545, shoulder=lefty, elbow=epositive, wrist=wpositive, fatherId=fReference[0]}
  [965] = {x=-207.187, y=39.932, z=154, rx=180, rz=102.273, shoulder=lefty, elbow=epositive, wrist=wpositive, fatherId=fReference[0]}
  [966] = {x=-205.052, y=49.745, z=154, rx=180, rz=105, shoulder=lefty, elbow=epositive, wrist=wpositive, fatherId=fReference[0]}
  [967] = {x=-202.453, y=59.446, z=154, rx=180, rz=107.727, shoulder=lefty, elbow=epositive, wrist=wpositive, fatherId=fReference[0]}
  [968] = {x=-199.395, y=69.011, z=154, rx=180, rz=110.455, shoulder=lefty, elbow=epositive, wrist=wpositive, fatherId=fReference[0]}
  [969] = {x=-195.886, y=78.421, z=154, rx=180, rz=113.182, shoulder=lefty, elbow=epositive, wrist=wpositive, fatherId=fReference[0]}
  [970] = {x=-191.932, y=87.653, z=154, rx=180, rz=115.909, shoulder=lefty, elbow=epositive, wrist=wpositive, fatherId=fReference[0]}
  [971] = {x=-187.544, y=96.686, z=154, rx=180, rz=118.636, shoulder=lefty, elbow=epositive, wrist=wpositive, fatherId=fReference[0]}
  [972] = {x=-182.731, y=105.5, z=154, rx=180, rz=121.364, shoulder=lefty, elbow=epositive, wrist=wpositive, fatherId=fReference[0]}
  [973] = {x=-177.505, y=114.075, z=154, rx=180, rz=124.091, shoulder=lefty, elbow=epositive, wrist=wpositive, fatherId=fReference[0]}
  [974] = {x=-171.876, y=122.392, z=154, rx=180, rz=126.818, shoulder=lefty, elbow=epositive, wrist=wpositive, fatherId=fReference[0]}
  [975] = {x=-165.857, y=130.432, z=154, rx=180, rz=129.545, shoulder=lefty, elbow=epositive, wrist=wpositive, fatherId=fReference[0]}
  [976] = {x=-159.463, y=138.176, z=154, rx=180, rz=132.273, shoulder=lefty, elbow=epositive, wrist=wpositive, fatherId=fReference[0]}
  [977] = {x=-152.708, y=145.607, z=154, rx=-180, rz=135, shoulder=lefty, elbow=epositive, wrist=wpositive, fatherId=fReference[0]}
  [978] = {x=-145.607, y=152.708, z=154, rx=-180, rz=137.727, shoulder=lefty, elbow=epositive, wrist=wpositive, fatherId=fReference[0]}
  [979] = {x=-138.176, y=159.463, z=154, rx=180, rz=140.455, shoulder=lefty, elbow=epositive, wrist=wpositive, fatherId=fReference[0]}
  [980] = {x=-130.432, y=165.857, z=154, rx=180, rz=143.182, shoulder=lefty, elbow=epositive, wrist=wpositive, fatherId=fReference[0]}
  [981] = {x=-122.392, y=171.876, z=154, rx=180, rz=145.909, shoulder=lefty, elbow=epositive, wrist=wpositive, fatherId=fReference[0]}
  [982] = {x=-114.075, y=177.505, z=154, rx=180, rz=148.636, shoulder=lefty, elbow=epositive, wrist=wpositive, fatherId=fReference[0]}
  [983] = {x=-105.5, y=182.731, z=154, rx=180, rz=151.364, shoulder=lefty, elbow=epositive, wrist=wpositive, fatherId=fReference[0]}
  [984] = {x=-96.686, y=187.544, z=154, rx=-180, rz=154.091, shoulder=lefty, elbow=epositive, wrist=wpositive, fatherId=fReference[0]}
  [985] = {x=-87.653, y=191.932, z=154, rx=-180, rz=156.818, shoulder=lefty, elbow=epositive, wrist=wpositive, fatherId=fReference[0]}
  [986] = {x=-78.421, y=195.886, z=154, rx=180, rz=159.545, shoulder=lefty, elbow=epositive, wrist=wpositive, fatherId=fReference[0]}
  [987] = {x=-69.011, y=199.395, z=154, rx=-180, rz=162.273, shoulder=lefty, elbow=epositive, wrist=wpositive, fatherId=fReference[0]}
  [988] = {x=-59.446, y=202.453, z=154, rx=180, rz=165, shoulder=lefty, elbow=epositive, wrist=wpositive, fatherId=fReference[0]}
  [989] = {x=-49.745, y=205.052, z=154, rx=180, rz=167.727, shoulder=lefty, elbow=epositive, wrist=wpositive, fatherId=fReference[0]}
  [990] = {x=-39.932, y=207.187, z=154, rx=180, rz=170.455, shoulder=lefty, elbow=epositive, wrist=wpositive, fatherId=fReference[0]}
  [991] = {x=-30.028, y=208.852, z=154, rx=-180, rz=173.182, shoulder=lefty, elbow=epositive, wrist=wpositive, fatherId=fReference[0]}
  [992] = {x=-20.057, y=210.045, z=154, rx=-180, rz=175.909, shoulder=lefty, elbow=epositive, wrist=wpositive, fatherId=fReference[0]}
  [993] = {x=-10.04, y=210.761, z=154, rx=-180, rz=178.636, shoulder=lefty, elbow=epositive, wrist=wpositive, fatherId=fReference[0]}
  [994] = {y=211, z=154, rx=-180, rz=-178.636, shoulder=lefty, elbow=epositive, wrist=wpositive, fatherId=fReference[0]}
  [995] = {x=10.04, y=210.761, z=154, rx=180, rz=-175.909, shoulder=lefty, elbow=epositive, wrist=wpositive, fatherId=fReference[0]}
  [996] = {x=20.057, y=210.045, z=154, rx=-180, rz=-173.182, shoulder=lefty, elbow=epositive, wrist=wpositive, fatherId=fReference[0]}
  [997] = {x=30.028, y=208.852, z=154, rx=-180, rz=-170.455, shoulder=lefty, elbow=epositive, wrist=wpositive, fatherId=fReference[0]}
  [998] = {x=39.932, y=207.187, z=154, rx=-180, rz=-167.727, shoulder=lefty, elbow=epositive, wrist=wpositive, fatherId=fReference[0]}
  [999] = {x=49.745, y=205.052, z=154, rx=-180, rz=-165, shoulder=lefty, elbow=epositive, wrist=wpositive, fatherId=fReference[0]}
  [1000] = {x=59.446, y=202.453, z=154, rx=-180, rz=-162.273, shoulder=lefty, elbow=epositive, wrist=wpositive, fatherId=fReference[0]}
  [1001] = {x=69.011, y=199.395, z=154, rx=-180, rz=-159.545, shoulder=lefty, elbow=epositive, wrist=wpositive, fatherId=fReference[0]}
  [1002] = {x=78.421, y=195.886, z=154, rx=-180, rz=-156.818, shoulder=lefty, elbow=epositive, wrist=wpositive, fatherId=fReference[0]}
  [1003] = {x=87.653, y=191.932, z=154, rx=180, rz=-154.091, shoulder=lefty, elbow=epositive, wrist=wpositive, fatherId=fReference[0]}
  [1004] = {x=96.686, y=187.544, z=154, rx=-180, rz=-151.364, shoulder=lefty, elbow=epositive, wrist=wpositive, fatherId=fReference[0]}
  [1005] = {x=105.5, y=182.731, z=154, rx=-180, rz=-148.636, shoulder=lefty, elbow=epositive, wrist=wpositive, fatherId=fReference[0]}
  [1006] = {x=114.075, y=177.505, z=154, rx=-180, rz=-145.909, shoulder=lefty, elbow=epositive, wrist=wpositive, fatherId=fReference[0]}
  [1007] = {x=122.392, y=171.876, z=154, rx=-180, rz=-143.182, shoulder=lefty, elbow=epositive, wrist=wpositive, fatherId=fReference[0]}
  [1008] = {x=130.432, y=165.857, z=154, rx=-180, rz=-140.455, shoulder=lefty, elbow=epositive, wrist=wpositive, fatherId=fReference[0]}
  [1009] = {x=138.176, y=159.463, z=154, rx=-180, rz=-137.727, shoulder=lefty, elbow=epositive, wrist=wpositive, fatherId=fReference[0]}
  [1010] = {x=145.607, y=152.708, z=154, rx=-180, rz=-135, shoulder=lefty, elbow=epositive, wrist=wpositive, fatherId=fReference[0]}
  [1011] = {x=152.708, y=145.607, z=154, rx=-180, rz=-132.273, shoulder=lefty, elbow=epositive, wrist=wpositive, fatherId=fReference[0]}
  [1012] = {x=159.463, y=138.176, z=154, rx=-180, rz=-129.545, shoulder=lefty, elbow=epositive, wrist=wpositive, fatherId=fReference[0]}
  [1013] = {x=165.857, y=130.432, z=154, rx=-180, rz=-126.818, shoulder=lefty, elbow=epositive, wrist=wpositive, fatherId=fReference[0]}
  [1014] = {x=171.876, y=122.392, z=154, rx=-180, rz=-124.091, shoulder=lefty, elbow=epositive, wrist=wpositive, fatherId=fReference[0]}
  [1015] = {x=177.505, y=114.075, z=154, rx=-180, rz=-121.364, shoulder=lefty, elbow=epositive, wrist=wpositive, fatherId=fReference[0]}
  [1016] = {x=182.731, y=105.5, z=154, rx=-180, rz=-118.636, shoulder=lefty, elbow=epositive, wrist=wpositive, fatherId=fReference[0]}
  [1017] = {x=187.544, y=96.686, z=154, rx=-180, rz=-115.909, shoulder=lefty, elbow=epositive, wrist=wpositive, fatherId=fReference[0]}
  [1018] = {x=191.932, y=87.653, z=154, rx=-180, rz=-113.182, shoulder=lefty, elbow=epositive, wrist=wpositive, fatherId=fReference[0]}
  [1019] = {x=195.886, y=78.421, z=154, rx=-180, rz=-110.455, shoulder=lefty, elbow=epositive, wrist=wpositive, fatherId=fReference[0]}
  [1020] = {x=199.395, y=69.011, z=154, rx=-180, rz=-107.727, shoulder=lefty, elbow=epositive, wrist=wpositive, fatherId=fReference[0]}
  [1021] = {x=202.453, y=59.446, z=154, rx=-180, rz=-105, shoulder=lefty, elbow=epositive, wrist=wpositive, fatherId=fReference[0]}
  [1022] = {x=205.052, y=49.745, z=154, rx=-180, rz=-102.273, shoulder=lefty, elbow=epositive, wrist=wpositive, fatherId=fReference[0]}
  [1023] = {x=207.187, y=39.932, z=154, rx=-180, rz=-99.545, shoulder=lefty, elbow=epositive, wrist=wpositive, fatherId=fReference[0]}
  [1024] = {x=208.852, y=30.028, z=154, rx=-180, rz=-96.818, shoulder=lefty, elbow=epositive, wrist=wpositive, fatherId=fReference[0]}
  [1025] = {x=210.045, y=20.057, z=154, rx=-180, rz=-94.091, shoulder=lefty, elbow=epositive, wrist=wpositive, fatherId=fReference[0]}
  [1026] = {x=210.761, y=10.04, z=154, rx=-180, rz=-91.364, shoulder=lefty, elbow=epositive, wrist=wpositive, fatherId=fReference[0]}
  [1027] = {x=211, z=154, rx=180, rz=-88.636, shoulder=lefty, elbow=epositive, wrist=wpositive, fatherId=fReference[0]}
  [1028] = {x=210.761, y=-10.04, z=154, rx=180, rz=-85.909, shoulder=lefty, elbow=epositive, wrist=wpositive, fatherId=fReference[0]}
  [1029] = {x=210.045, y=-20.057, z=154, rx=180, rz=-83.182, shoulder=lefty, elbow=epositive, wrist=wpositive, fatherId=fReference[0]}
  [1030] = {x=208.852, y=-30.028, z=154, rx=180, rz=-80.455, shoulder=lefty, elbow=epositive, wrist=wpositive, fatherId=fReference[0]}
  [1031] = {x=207.187, y=-39.932, z=154, rx=-180, rz=-77.727, shoulder=lefty, elbow=epositive, wrist=wpositive, fatherId=fReference[0]}
  [1032] = {x=205.052, y=-49.745, z=154, rx=180, rz=-75, shoulder=lefty, elbow=epositive, wrist=wpositive, fatherId=fReference[0]}
  [1033] = {x=202.453, y=-59.446, z=154, rx=180, rz=-72.273, shoulder=lefty, elbow=epositive, wrist=wpositive, fatherId=fReference[0]}
  [1034] = {x=199.395, y=-69.011, z=154, rx=180, rz=-69.545, shoulder=lefty, elbow=epositive, wrist=wpositive, fatherId=fReference[0]}
  [1035] = {x=195.886, y=-78.421, z=154, rx=-180, rz=-66.818, shoulder=lefty, elbow=epositive, wrist=wpositive, fatherId=fReference[0]}
  [1036] = {x=191.932, y=-87.653, z=154, rx=180, rz=-64.091, shoulder=lefty, elbow=epositive, wrist=wpositive, fatherId=fReference[0]}
  [1037] = {x=187.544, y=-96.686, z=154, rx=180, rz=-61.364, shoulder=lefty, elbow=epositive, wrist=wpositive, fatherId=fReference[0]}
  [1038] = {x=182.731, y=-105.5, z=154, rx=180, rz=-58.636, shoulder=lefty, elbow=epositive, wrist=wpositive, fatherId=fReference[0]}
  [1039] = {x=177.505, y=-114.075, z=154, rx=-180, rz=-55.909, shoulder=lefty, elbow=epositive, wrist=wpositive, fatherId=fReference[0]}
  [1040] = {x=171.876, y=-122.392, z=154, rx=-180, rz=-53.182, shoulder=lefty, elbow=epositive, wrist=wpositive, fatherId=fReference[0]}
  [1041] = {x=165.857, y=-130.432, z=154, rx=180, rz=-50.455, shoulder=lefty, elbow=epositive, wrist=wpositive, fatherId=fReference[0]}
  [1042] = {x=159.463, y=-138.176, z=154, rx=180, rz=-47.727, shoulder=lefty, elbow=epositive, wrist=wpositive, fatherId=fReference[0]}
  [1043] = {x=152.708, y=-145.607, z=154, rx=-180, rz=-45, shoulder=lefty, elbow=epositive, wrist=wpositive, fatherId=fReference[0]}
  [1044] = {x=145.607, y=-152.708, z=154, rx=180, rz=-42.273, shoulder=lefty, elbow=epositive, wrist=wpositive, fatherId=fReference[0]}
  [1045] = {x=138.176, y=-159.463, z=154, rx=180, rz=-39.545, shoulder=lefty, elbow=epositive, wrist=wpositive, fatherId=fReference[0]}
  [1046] = {x=130.432, y=-165.857, z=154, rx=180, rz=-36.818, shoulder=lefty, elbow=epositive, wrist=wpositive, fatherId=fReference[0]}
  [1047] = {x=122.392, y=-171.876, z=154, rx=180, rz=-34.091, shoulder=lefty, elbow=epositive, wrist=wpositive, fatherId=fReference[0]}
  [1048] = {x=114.075, y=-177.505, z=154, rx=180, rz=-31.364, shoulder=lefty, elbow=epositive, wrist=wpositive, fatherId=fReference[0]}
  [1049] = {x=105.5, y=-182.731, z=154, rx=180, rz=-28.636, shoulder=lefty, elbow=epositive, wrist=wpositive, fatherId=fReference[0]}
  [1050] = {x=96.686, y=-187.544, z=154, rx=180, rz=-25.909, shoulder=lefty, elbow=epositive, wrist=wpositive, fatherId=fReference[0]}
  [1051] = {x=87.653, y=-191.932, z=154, rx=180, rz=-23.182, shoulder=lefty, elbow=epositive, wrist=wpositive, fatherId=fReference[0]}
  [1052] = {x=78.421, y=-195.886, z=154, rx=-180, rz=-20.455, shoulder=lefty, elbow=epositive, wrist=wpositive, fatherId=fReference[0]}
  [1053] = {x=69.011, y=-199.395, z=154, rx=-180, rz=-17.727, shoulder=lefty, elbow=epositive, wrist=wpositive, fatherId=fReference[0]}
  [1054] = {x=59.446, y=-202.453, z=154, rx=180, rz=-15, shoulder=lefty, elbow=epositive, wrist=wpositive, fatherId=fReference[0]}
  [1055] = {x=49.745, y=-205.052, z=154, rx=180, rz=-12.273, shoulder=lefty, elbow=epositive, wrist=wpositive, fatherId=fReference[0]}
  [1056] = {x=39.932, y=-207.187, z=154, rx=180, rz=-9.545, shoulder=lefty, elbow=epositive, wrist=wpositive, fatherId=fReference[0]}
  [1057] = {x=30.028, y=-208.852, z=154, rx=-180, rz=-6.818, shoulder=lefty, elbow=epositive, wrist=wpositive, fatherId=fReference[0]}
  [1058] = {x=20.057, y=-210.045, z=154, rx=-180, rz=-4.091, shoulder=lefty, elbow=epositive, wrist=wpositive, fatherId=fReference[0]}
  [1059] = {x=10.04, y=-210.761, z=154, rx=-180, rz=-1.364, shoulder=lefty, elbow=epositive, wrist=wpositive, fatherId=fReference[0]}
  [1060] = {y=-211, z=154, rx=-180, rz=1.364, shoulder=lefty, elbow=epositive, wrist=wpositive, fatherId=fReference[0]}
  [1061] = {x=-10.04, y=-210.761, z=154, rx=-180, rz=4.091, shoulder=lefty, elbow=epositive, wrist=wpositive, fatherId=fReference[0]}
  [1062] = {x=-20.057, y=-210.045, z=154, rx=-180, rz=6.818, shoulder=lefty, elbow=epositive, wrist=wpositive, fatherId=fReference[0]}
  [1063] = {x=-30.028, y=-208.852, z=154, rx=-180, rz=9.545, shoulder=lefty, elbow=epositive, wrist=wpositive, fatherId=fReference[0]}
  [1064] = {x=-39.932, y=-207.187, z=154, rx=180, rz=12.273, shoulder=lefty, elbow=epositive, wrist=wpositive, fatherId=fReference[0]}
  [1065] = {x=-49.745, y=-205.052, z=154, rx=-180, rz=15, shoulder=lefty, elbow=epositive, wrist=wpositive, fatherId=fReference[0]}
  [1066] = {x=-59.446, y=-202.453, z=154, rx=180, rz=17.727, shoulder=lefty, elbow=epositive, wrist=wpositive, fatherId=fReference[0]}
  [1067] = {x=-69.011, y=-199.395, z=154, rx=180, rz=20.455, shoulder=lefty, elbow=epositive, wrist=wpositive, fatherId=fReference[0]}
  [1068] = {x=-78.421, y=-195.886, z=154, rx=-180, rz=23.182, shoulder=lefty, elbow=epositive, wrist=wpositive, fatherId=fReference[0]}
  [1069] = {x=-87.653, y=-191.932, z=154, rx=-180, rz=25.909, shoulder=lefty, elbow=epositive, wrist=wpositive, fatherId=fReference[0]}
  [1070] = {x=-96.686, y=-187.544, z=154, rx=-180, rz=28.636, shoulder=lefty, elbow=epositive, wrist=wpositive, fatherId=fReference[0]}
  [1071] = {x=-105.5, y=-182.731, z=154, rx=-180, rz=31.364, shoulder=lefty, elbow=epositive, wrist=wpositive, fatherId=fReference[0]}
  [1072] = {x=-114.075, y=-177.505, z=154, rx=-180, rz=34.091, shoulder=lefty, elbow=epositive, wrist=wpositive, fatherId=fReference[0]}
  [1073] = {x=-122.392, y=-171.876, z=154, rx=-180, rz=36.818, shoulder=lefty, elbow=epositive, wrist=wpositive, fatherId=fReference[0]}
  [1074] = {x=-130.432, y=-165.857, z=154, rx=180, rz=39.545, shoulder=lefty, elbow=epositive, wrist=wpositive, fatherId=fReference[0]}
  [1075] = {x=-138.176, y=-159.463, z=154, rx=-180, rz=42.273, shoulder=lefty, elbow=epositive, wrist=wpositive, fatherId=fReference[0]}
  [1076] = {x=-145.607, y=-152.708, z=154, rx=-180, rz=45, shoulder=lefty, elbow=epositive, wrist=wpositive, fatherId=fReference[0]}
  [1077] = {x=-152.708, y=-145.607, z=154, rx=-180, rz=47.727, shoulder=lefty, elbow=epositive, wrist=wpositive, fatherId=fReference[0]}
  [1078] = {x=-159.463, y=-138.176, z=154, rx=-180, rz=50.455, shoulder=lefty, elbow=epositive, wrist=wpositive, fatherId=fReference[0]}
  [1079] = {x=-165.857, y=-130.432, z=154, rx=-180, rz=53.182, shoulder=lefty, elbow=epositive, wrist=wpositive, fatherId=fReference[0]}
  [1080] = {x=-171.876, y=-122.392, z=154, rx=-180, rz=55.909, shoulder=lefty, elbow=epositive, wrist=wpositive, fatherId=fReference[0]}
  [1081] = {x=-177.505, y=-114.075, z=154, rx=-180, rz=58.636, shoulder=lefty, elbow=epositive, wrist=wpositive, fatherId=fReference[0]}
  [1082] = {x=-182.731, y=-105.5, z=154, rx=-180, rz=61.364, shoulder=lefty, elbow=epositive, wrist=wpositive, fatherId=fReference[0]}
  [1083] = {x=-187.544, y=-96.686, z=154, rx=-180, rz=64.091, shoulder=lefty, elbow=epositive, wrist=wpositive, fatherId=fReference[0]}
  [1084] = {x=-191.932, y=-87.653, z=154, rx=-180, rz=66.818, shoulder=lefty, elbow=epositive, wrist=wpositive, fatherId=fReference[0]}
  [1085] = {x=-195.886, y=-78.421, z=154, rx=-180, rz=69.545, shoulder=lefty, elbow=epositive, wrist=wpositive, fatherId=fReference[0]}
  [1086] = {x=-199.395, y=-69.011, z=154, rx=-180, rz=72.273, shoulder=lefty, elbow=epositive, wrist=wpositive, fatherId=fReference[0]}
  [1087] = {x=-202.453, y=-59.446, z=154, rx=-180, rz=75, shoulder=lefty, elbow=epositive, wrist=wpositive, fatherId=fReference[0]}
  [1088] = {x=-205.052, y=-49.745, z=154, rx=-180, rz=77.727, shoulder=lefty, elbow=epositive, wrist=wpositive, fatherId=fReference[0]}
  [1089] = {x=-207.187, y=-39.932, z=154, rx=-180, rz=80.455, shoulder=lefty, elbow=epositive, wrist=wpositive, fatherId=fReference[0]}
  [1090] = {x=-208.852, y=-30.028, z=154, rx=-180, rz=83.182, shoulder=lefty, elbow=epositive, wrist=wpositive, fatherId=fReference[0]}
  [1091] = {x=-210.045, y=-20.057, z=154, rx=-180, rz=85.909, shoulder=lefty, elbow=epositive, wrist=wpositive, fatherId=fReference[0]}
  [1092] = {x=-210.761, y=-10.04, z=154, rx=-180, rz=88.636, shoulder=lefty, elbow=epositive, wrist=wpositive, fatherId=fReference[0]}
  [1093] = {x=-211, z=154, rx=-180, rz=88.636, shoulder=lefty, elbow=epositive, wrist=wpositive, fatherId=fReference[0]}
  [1094] = {x=-211, z=154, rx=-180, rz=88.636, shoulder=lefty, elbow=epositive, wrist=wpositive, fatherId=fReference[0]}
  [1095] = {x=-211, z=254, rx=-180, rz=88.636, shoulder=lefty, elbow=epositive, wrist=wpositive, fatherId=fReference[0]}
  [1096] = {x=-211, z=276, rx=-180, rz=88.636, shoulder=lefty, elbow=epositive, wrist=wpositive, fatherId=fReference[0]}
  [1097] = {x=-211, z=176, rx=-180, rz=88.636, shoulder=lefty, elbow=epositive, wrist=wpositive, fatherId=fReference[0]}
  [1098] = {x=-211, z=176, rx=-180, rz=88.636, shoulder=lefty, elbow=epositive, wrist=wpositive, fatherId=fReference[0]}
  [1099] = {x=-210.761, y=-10.04, z=176, rx=-180, rz=85.909, shoulder=lefty, elbow=epositive, wrist=wpositive, fatherId=fReference[0]}
  [1100] = {x=-210.045, y=-20.057, z=176, rx=-180, rz=83.182, shoulder=lefty, elbow=epositive, wrist=wpositive, fatherId=fReference[0]}
  [1101] = {x=-208.852, y=-30.028, z=176, rx=-180, rz=80.455, shoulder=lefty, elbow=epositive, wrist=wpositive, fatherId=fReference[0]}
  [1102] = {x=-207.187, y=-39.932, z=176, rx=-180, rz=77.727, shoulder=lefty, elbow=epositive, wrist=wpositive, fatherId=fReference[0]}
  [1103] = {x=-205.052, y=-49.745, z=176, rx=-180, rz=75, shoulder=lefty, elbow=epositive, wrist=wpositive, fatherId=fReference[0]}
  [1104] = {x=-202.453, y=-59.446, z=176, rx=180, rz=72.273, shoulder=lefty, elbow=epositive, wrist=wpositive, fatherId=fReference[0]}
  [1105] = {x=-199.395, y=-69.011, z=176, rx=-180, rz=69.545, shoulder=lefty, elbow=epositive, wrist=wpositive, fatherId=fReference[0]}
  [1106] = {x=-195.886, y=-78.421, z=176, rx=-180, rz=66.818, shoulder=lefty, elbow=epositive, wrist=wpositive, fatherId=fReference[0]}
  [1107] = {x=-191.932, y=-87.653, z=176, rx=-180, rz=64.091, shoulder=lefty, elbow=epositive, wrist=wpositive, fatherId=fReference[0]}
  [1108] = {x=-187.544, y=-96.686, z=176, rx=180, rz=61.364, shoulder=lefty, elbow=epositive, wrist=wpositive, fatherId=fReference[0]}
  [1109] = {x=-182.731, y=-105.5, z=176, rx=180, rz=58.636, shoulder=lefty, elbow=epositive, wrist=wpositive, fatherId=fReference[0]}
  [1110] = {x=-177.505, y=-114.075, z=176, rx=-180, rz=55.909, shoulder=lefty, elbow=epositive, wrist=wpositive, fatherId=fReference[0]}
  [1111] = {x=-171.876, y=-122.392, z=176, rx=-180, rz=53.182, shoulder=lefty, elbow=epositive, wrist=wpositive, fatherId=fReference[0]}
  [1112] = {x=-165.857, y=-130.432, z=176, rx=-180, rz=50.455, shoulder=lefty, elbow=epositive, wrist=wpositive, fatherId=fReference[0]}
  [1113] = {x=-159.463, y=-138.176, z=176, rx=-180, rz=47.727, shoulder=lefty, elbow=epositive, wrist=wpositive, fatherId=fReference[0]}
  [1114] = {x=-152.708, y=-145.607, z=176, rx=-180, rz=45, shoulder=lefty, elbow=epositive, wrist=wpositive, fatherId=fReference[0]}
  [1115] = {x=-145.607, y=-152.708, z=176, rx=180, rz=42.273, shoulder=lefty, elbow=epositive, wrist=wpositive, fatherId=fReference[0]}
  [1116] = {x=-138.176, y=-159.463, z=176, rx=-180, rz=39.545, shoulder=lefty, elbow=epositive, wrist=wpositive, fatherId=fReference[0]}
  [1117] = {x=-130.432, y=-165.857, z=176, rx=-180, rz=36.818, shoulder=lefty, elbow=epositive, wrist=wpositive, fatherId=fReference[0]}
  [1118] = {x=-122.392, y=-171.876, z=176, rx=-180, rz=34.091, shoulder=lefty, elbow=epositive, wrist=wpositive, fatherId=fReference[0]}
  [1119] = {x=-114.075, y=-177.505, z=176, rx=-180, rz=31.364, shoulder=lefty, elbow=epositive, wrist=wpositive, fatherId=fReference[0]}
  [1120] = {x=-105.5, y=-182.731, z=176, rx=-180, rz=28.636, shoulder=lefty, elbow=epositive, wrist=wpositive, fatherId=fReference[0]}
  [1121] = {x=-96.686, y=-187.544, z=176, rx=180, rz=25.909, shoulder=lefty, elbow=epositive, wrist=wpositive, fatherId=fReference[0]}
  [1122] = {x=-87.653, y=-191.932, z=176, rx=180, rz=23.182, shoulder=lefty, elbow=epositive, wrist=wpositive, fatherId=fReference[0]}
  [1123] = {x=-78.421, y=-195.886, z=176, rx=-180, rz=20.455, shoulder=lefty, elbow=epositive, wrist=wpositive, fatherId=fReference[0]}
  [1124] = {x=-69.011, y=-199.395, z=176, rx=180, rz=17.727, shoulder=lefty, elbow=epositive, wrist=wpositive, fatherId=fReference[0]}
  [1125] = {x=-59.446, y=-202.453, z=176, rx=-180, rz=15, shoulder=lefty, elbow=epositive, wrist=wpositive, fatherId=fReference[0]}
  [1126] = {x=-49.745, y=-205.052, z=176, rx=-180, rz=12.273, shoulder=lefty, elbow=epositive, wrist=wpositive, fatherId=fReference[0]}
  [1127] = {x=-39.932, y=-207.187, z=176, rx=-180, rz=9.545, shoulder=lefty, elbow=epositive, wrist=wpositive, fatherId=fReference[0]}
  [1128] = {x=-30.028, y=-208.852, z=176, rx=180, rz=6.818, shoulder=lefty, elbow=epositive, wrist=wpositive, fatherId=fReference[0]}
  [1129] = {x=-20.057, y=-210.045, z=176, rx=180, rz=4.091, shoulder=lefty, elbow=epositive, wrist=wpositive, fatherId=fReference[0]}
  [1130] = {x=-10.04, y=-210.761, z=176, rx=180, rz=1.364, shoulder=lefty, elbow=epositive, wrist=wpositive, fatherId=fReference[0]}
  [1131] = {y=-211, z=176, rx=-180, rz=-1.364, shoulder=lefty, elbow=epositive, wrist=wpositive, fatherId=fReference[0]}
  [1132] = {x=10.04, y=-210.761, z=176, rx=-180, rz=-4.091, shoulder=lefty, elbow=epositive, wrist=wpositive, fatherId=fReference[0]}
  [1133] = {x=20.057, y=-210.045, z=176, rx=-180, rz=-6.818, shoulder=lefty, elbow=epositive, wrist=wpositive, fatherId=fReference[0]}
  [1134] = {x=30.028, y=-208.852, z=176, rx=-180, rz=-9.545, shoulder=lefty, elbow=epositive, wrist=wpositive, fatherId=fReference[0]}
  [1135] = {x=39.932, y=-207.187, z=176, rx=180, rz=-12.273, shoulder=lefty, elbow=epositive, wrist=wpositive, fatherId=fReference[0]}
  [1136] = {x=49.745, y=-205.052, z=176, rx=-180, rz=-15, shoulder=lefty, elbow=epositive, wrist=wpositive, fatherId=fReference[0]}
  [1137] = {x=59.446, y=-202.453, z=176, rx=180, rz=-17.727, shoulder=lefty, elbow=epositive, wrist=wpositive, fatherId=fReference[0]}
  [1138] = {x=69.011, y=-199.395, z=176, rx=-180, rz=-20.455, shoulder=lefty, elbow=epositive, wrist=wpositive, fatherId=fReference[0]}
  [1139] = {x=78.421, y=-195.886, z=176, rx=180, rz=-23.182, shoulder=lefty, elbow=epositive, wrist=wpositive, fatherId=fReference[0]}
  [1140] = {x=87.653, y=-191.932, z=176, rx=180, rz=-25.909, shoulder=lefty, elbow=epositive, wrist=wpositive, fatherId=fReference[0]}
  [1141] = {x=96.686, y=-187.544, z=176, rx=-180, rz=-28.636, shoulder=lefty, elbow=epositive, wrist=wpositive, fatherId=fReference[0]}
  [1142] = {x=105.5, y=-182.731, z=176, rx=180, rz=-31.364, shoulder=lefty, elbow=epositive, wrist=wpositive, fatherId=fReference[0]}
  [1143] = {x=114.075, y=-177.505, z=176, rx=-180, rz=-34.091, shoulder=lefty, elbow=epositive, wrist=wpositive, fatherId=fReference[0]}
  [1144] = {x=122.392, y=-171.876, z=176, rx=-180, rz=-36.818, shoulder=lefty, elbow=epositive, wrist=wpositive, fatherId=fReference[0]}
  [1145] = {x=130.432, y=-165.857, z=176, rx=180, rz=-39.545, shoulder=lefty, elbow=epositive, wrist=wpositive, fatherId=fReference[0]}
  [1146] = {x=138.176, y=-159.463, z=176, rx=180, rz=-42.273, shoulder=lefty, elbow=epositive, wrist=wpositive, fatherId=fReference[0]}
  [1147] = {x=145.607, y=-152.708, z=176, rx=180, rz=-45, shoulder=lefty, elbow=epositive, wrist=wpositive, fatherId=fReference[0]}
  [1148] = {x=152.708, y=-145.607, z=176, rx=180, rz=-47.727, shoulder=lefty, elbow=epositive, wrist=wpositive, fatherId=fReference[0]}
  [1149] = {x=159.463, y=-138.176, z=176, rx=180, rz=-50.455, shoulder=lefty, elbow=epositive, wrist=wpositive, fatherId=fReference[0]}
  [1150] = {x=165.857, y=-130.432, z=176, rx=180, rz=-53.182, shoulder=lefty, elbow=epositive, wrist=wpositive, fatherId=fReference[0]}
  [1151] = {x=171.876, y=-122.392, z=176, rx=-180, rz=-55.909, shoulder=lefty, elbow=epositive, wrist=wpositive, fatherId=fReference[0]}
  [1152] = {x=177.505, y=-114.075, z=176, rx=180, rz=-58.636, shoulder=lefty, elbow=epositive, wrist=wpositive, fatherId=fReference[0]}
  [1153] = {x=182.731, y=-105.5, z=176, rx=180, rz=-61.364, shoulder=lefty, elbow=epositive, wrist=wpositive, fatherId=fReference[0]}
  [1154] = {x=187.544, y=-96.686, z=176, rx=180, rz=-64.091, shoulder=lefty, elbow=epositive, wrist=wpositive, fatherId=fReference[0]}
  [1155] = {x=191.932, y=-87.653, z=176, rx=180, rz=-66.818, shoulder=lefty, elbow=epositive, wrist=wpositive, fatherId=fReference[0]}
  [1156] = {x=195.886, y=-78.421, z=176, rx=180, rz=-69.545, shoulder=lefty, elbow=epositive, wrist=wpositive, fatherId=fReference[0]}
  [1157] = {x=199.395, y=-69.011, z=176, rx=180, rz=-72.273, shoulder=lefty, elbow=epositive, wrist=wpositive, fatherId=fReference[0]}
  [1158] = {x=202.453, y=-59.446, z=176, rx=180, rz=-75, shoulder=lefty, elbow=epositive, wrist=wpositive, fatherId=fReference[0]}
  [1159] = {x=205.052, y=-49.745, z=176, rx=180, rz=-77.727, shoulder=lefty, elbow=epositive, wrist=wpositive, fatherId=fReference[0]}
  [1160] = {x=207.187, y=-39.932, z=176, rx=-180, rz=-80.455, shoulder=lefty, elbow=epositive, wrist=wpositive, fatherId=fReference[0]}
  [1161] = {x=208.852, y=-30.028, z=176, rx=180, rz=-83.182, shoulder=lefty, elbow=epositive, wrist=wpositive, fatherId=fReference[0]}
  [1162] = {x=210.045, y=-20.057, z=176, rx=180, rz=-85.909, shoulder=lefty, elbow=epositive, wrist=wpositive, fatherId=fReference[0]}
  [1163] = {x=210.761, y=-10.04, z=176, rx=180, rz=-88.636, shoulder=lefty, elbow=epositive, wrist=wpositive, fatherId=fReference[0]}
  [1164] = {x=211, z=176, rx=-180, rz=-91.364, shoulder=lefty, elbow=epositive, wrist=wpositive, fatherId=fReference[0]}
  [1165] = {x=210.761, y=10.04, z=176, rx=-180, rz=-94.091, shoulder=lefty, elbow=epositive, wrist=wpositive, fatherId=fReference[0]}
  [1166] = {x=210.045, y=20.057, z=176, rx=-180, rz=-96.818, shoulder=lefty, elbow=epositive, wrist=wpositive, fatherId=fReference[0]}
  [1167] = {x=208.852, y=30.028, z=176, rx=-180, rz=-99.545, shoulder=lefty, elbow=epositive, wrist=wpositive, fatherId=fReference[0]}
  [1168] = {x=207.187, y=39.932, z=176, rx=-180, rz=-102.273, shoulder=lefty, elbow=epositive, wrist=wpositive, fatherId=fReference[0]}
  [1169] = {x=205.052, y=49.745, z=176, rx=-180, rz=-105, shoulder=lefty, elbow=epositive, wrist=wpositive, fatherId=fReference[0]}
  [1170] = {x=202.453, y=59.446, z=176, rx=-180, rz=-107.727, shoulder=lefty, elbow=epositive, wrist=wpositive, fatherId=fReference[0]}
  [1171] = {x=199.395, y=69.011, z=176, rx=-180, rz=-110.455, shoulder=lefty, elbow=epositive, wrist=wpositive, fatherId=fReference[0]}
  [1172] = {x=195.886, y=78.421, z=176, rx=-180, rz=-113.182, shoulder=lefty, elbow=epositive, wrist=wpositive, fatherId=fReference[0]}
  [1173] = {x=191.932, y=87.653, z=176, rx=-180, rz=-115.909, shoulder=lefty, elbow=epositive, wrist=wpositive, fatherId=fReference[0]}
  [1174] = {x=187.544, y=96.686, z=176, rx=-180, rz=-118.636, shoulder=lefty, elbow=epositive, wrist=wpositive, fatherId=fReference[0]}
  [1175] = {x=182.731, y=105.5, z=176, rx=-180, rz=-121.364, shoulder=lefty, elbow=epositive, wrist=wpositive, fatherId=fReference[0]}
  [1176] = {x=177.505, y=114.075, z=176, rx=-180, rz=-124.091, shoulder=lefty, elbow=epositive, wrist=wpositive, fatherId=fReference[0]}
  [1177] = {x=171.876, y=122.392, z=176, rx=-180, rz=-126.818, shoulder=lefty, elbow=epositive, wrist=wpositive, fatherId=fReference[0]}
  [1178] = {x=165.857, y=130.432, z=176, rx=-180, rz=-129.545, shoulder=lefty, elbow=epositive, wrist=wpositive, fatherId=fReference[0]}
  [1179] = {x=159.463, y=138.176, z=176, rx=-180, rz=-132.273, shoulder=lefty, elbow=epositive, wrist=wpositive, fatherId=fReference[0]}
  [1180] = {x=152.708, y=145.607, z=176, rx=-180, rz=-135, shoulder=lefty, elbow=epositive, wrist=wpositive, fatherId=fReference[0]}
  [1181] = {x=145.607, y=152.708, z=176, rx=-180, rz=-137.727, shoulder=lefty, elbow=epositive, wrist=wpositive, fatherId=fReference[0]}
  [1182] = {x=138.176, y=159.463, z=176, rx=-180, rz=-140.455, shoulder=lefty, elbow=epositive, wrist=wpositive, fatherId=fReference[0]}
  [1183] = {x=130.432, y=165.857, z=176, rx=180, rz=-143.182, shoulder=lefty, elbow=epositive, wrist=wpositive, fatherId=fReference[0]}
  [1184] = {x=122.392, y=171.876, z=176, rx=180, rz=-145.909, shoulder=lefty, elbow=epositive, wrist=wpositive, fatherId=fReference[0]}
  [1185] = {x=114.075, y=177.505, z=176, rx=-180, rz=-148.636, shoulder=lefty, elbow=epositive, wrist=wpositive, fatherId=fReference[0]}
  [1186] = {x=105.5, y=182.731, z=176, rx=-180, rz=-151.364, shoulder=lefty, elbow=epositive, wrist=wpositive, fatherId=fReference[0]}
  [1187] = {x=96.686, y=187.544, z=176, rx=-180, rz=-154.091, shoulder=lefty, elbow=epositive, wrist=wpositive, fatherId=fReference[0]}
  [1188] = {x=87.653, y=191.932, z=176, rx=180, rz=-156.818, shoulder=lefty, elbow=epositive, wrist=wpositive, fatherId=fReference[0]}
  [1189] = {x=78.421, y=195.886, z=176, rx=-180, rz=-159.545, shoulder=lefty, elbow=epositive, wrist=wpositive, fatherId=fReference[0]}
  [1190] = {x=69.011, y=199.395, z=176, rx=-180, rz=-162.273, shoulder=lefty, elbow=epositive, wrist=wpositive, fatherId=fReference[0]}
  [1191] = {x=59.446, y=202.453, z=176, rx=180, rz=-165, shoulder=lefty, elbow=epositive, wrist=wpositive, fatherId=fReference[0]}
  [1192] = {x=49.745, y=205.052, z=176, rx=-180, rz=-167.727, shoulder=lefty, elbow=epositive, wrist=wpositive, fatherId=fReference[0]}
  [1193] = {x=39.932, y=207.187, z=176, rx=-180, rz=-170.455, shoulder=lefty, elbow=epositive, wrist=wpositive, fatherId=fReference[0]}
  [1194] = {x=30.028, y=208.852, z=176, rx=180, rz=-173.182, shoulder=lefty, elbow=epositive, wrist=wpositive, fatherId=fReference[0]}
  [1195] = {x=20.057, y=210.045, z=176, rx=-180, rz=-175.909, shoulder=lefty, elbow=epositive, wrist=wpositive, fatherId=fReference[0]}
  [1196] = {x=10.04, y=210.761, z=176, rx=180, rz=-178.636, shoulder=lefty, elbow=epositive, wrist=wpositive, fatherId=fReference[0]}
  [1197] = {y=211, z=176, rx=-180, rz=178.636, shoulder=lefty, elbow=epositive, wrist=wpositive, fatherId=fReference[0]}
  [1198] = {x=-10.04, y=210.761, z=176, rx=-180, rz=175.909, shoulder=lefty, elbow=epositive, wrist=wpositive, fatherId=fReference[0]}
  [1199] = {x=-20.057, y=210.045, z=176, rx=180, rz=173.182, shoulder=lefty, elbow=epositive, wrist=wpositive, fatherId=fReference[0]}
  [1200] = {x=-30.028, y=208.852, z=176, rx=180, rz=170.455, shoulder=lefty, elbow=epositive, wrist=wpositive, fatherId=fReference[0]}
  [1201] = {x=-39.932, y=207.187, z=176, rx=180, rz=167.727, shoulder=lefty, elbow=epositive, wrist=wpositive, fatherId=fReference[0]}
  [1202] = {x=-49.745, y=205.052, z=176, rx=180, rz=165, shoulder=lefty, elbow=epositive, wrist=wpositive, fatherId=fReference[0]}
  [1203] = {x=-59.446, y=202.453, z=176, rx=-180, rz=162.273, shoulder=lefty, elbow=epositive, wrist=wpositive, fatherId=fReference[0]}
  [1204] = {x=-69.011, y=199.395, z=176, rx=-180, rz=159.545, shoulder=lefty, elbow=epositive, wrist=wpositive, fatherId=fReference[0]}
  [1205] = {x=-78.421, y=195.886, z=176, rx=180, rz=156.818, shoulder=lefty, elbow=epositive, wrist=wpositive, fatherId=fReference[0]}
  [1206] = {x=-87.653, y=191.932, z=176, rx=180, rz=154.091, shoulder=lefty, elbow=epositive, wrist=wpositive, fatherId=fReference[0]}
  [1207] = {x=-96.686, y=187.544, z=176, rx=-180, rz=151.364, shoulder=lefty, elbow=epositive, wrist=wpositive, fatherId=fReference[0]}
  [1208] = {x=-105.5, y=182.731, z=176, rx=180, rz=148.636, shoulder=lefty, elbow=epositive, wrist=wpositive, fatherId=fReference[0]}
  [1209] = {x=-114.075, y=177.505, z=176, rx=180, rz=145.909, shoulder=lefty, elbow=epositive, wrist=wpositive, fatherId=fReference[0]}
  [1210] = {x=-122.392, y=171.876, z=176, rx=180, rz=143.182, shoulder=lefty, elbow=epositive, wrist=wpositive, fatherId=fReference[0]}
  [1211] = {x=-130.432, y=165.857, z=176, rx=-180, rz=140.455, shoulder=lefty, elbow=epositive, wrist=wpositive, fatherId=fReference[0]}
  [1212] = {x=-138.176, y=159.463, z=176, rx=180, rz=137.727, shoulder=lefty, elbow=epositive, wrist=wpositive, fatherId=fReference[0]}
  [1213] = {x=-145.607, y=152.708, z=176, rx=180, rz=135, shoulder=lefty, elbow=epositive, wrist=wpositive, fatherId=fReference[0]}
  [1214] = {x=-152.708, y=145.607, z=176, rx=-180, rz=132.273, shoulder=lefty, elbow=epositive, wrist=wpositive, fatherId=fReference[0]}
  [1215] = {x=-159.463, y=138.176, z=176, rx=180, rz=129.545, shoulder=lefty, elbow=epositive, wrist=wpositive, fatherId=fReference[0]}
  [1216] = {x=-165.857, y=130.432, z=176, rx=180, rz=126.818, shoulder=lefty, elbow=epositive, wrist=wpositive, fatherId=fReference[0]}
  [1217] = {x=-171.876, y=122.392, z=176, rx=180, rz=124.091, shoulder=lefty, elbow=epositive, wrist=wpositive, fatherId=fReference[0]}
  [1218] = {x=-177.505, y=114.075, z=176, rx=180, rz=121.364, shoulder=lefty, elbow=epositive, wrist=wpositive, fatherId=fReference[0]}
  [1219] = {x=-182.731, y=105.5, z=176, rx=180, rz=118.636, shoulder=lefty, elbow=epositive, wrist=wpositive, fatherId=fReference[0]}
  [1220] = {x=-187.544, y=96.686, z=176, rx=180, rz=115.909, shoulder=lefty, elbow=epositive, wrist=wpositive, fatherId=fReference[0]}
  [1221] = {x=-191.932, y=87.653, z=176, rx=180, rz=113.182, shoulder=lefty, elbow=epositive, wrist=wpositive, fatherId=fReference[0]}
  [1222] = {x=-195.886, y=78.421, z=176, rx=180, rz=110.455, shoulder=lefty, elbow=epositive, wrist=wpositive, fatherId=fReference[0]}
  [1223] = {x=-199.395, y=69.011, z=176, rx=180, rz=107.727, shoulder=lefty, elbow=epositive, wrist=wpositive, fatherId=fReference[0]}
  [1224] = {x=-202.453, y=59.446, z=176, rx=180, rz=105, shoulder=lefty, elbow=epositive, wrist=wpositive, fatherId=fReference[0]}
  [1225] = {x=-205.052, y=49.745, z=176, rx=180, rz=102.273, shoulder=lefty, elbow=epositive, wrist=wpositive, fatherId=fReference[0]}
  [1226] = {x=-207.187, y=39.932, z=176, rx=180, rz=99.545, shoulder=lefty, elbow=epositive, wrist=wpositive, fatherId=fReference[0]}
  [1227] = {x=-208.852, y=30.028, z=176, rx=180, rz=96.818, shoulder=lefty, elbow=epositive, wrist=wpositive, fatherId=fReference[0]}
  [1228] = {x=-210.045, y=20.057, z=176, rx=180, rz=94.091, shoulder=lefty, elbow=epositive, wrist=wpositive, fatherId=fReference[0]}
  [1229] = {x=-210.761, y=10.04, z=176, rx=180, rz=91.364, shoulder=lefty, elbow=epositive, wrist=wpositive, fatherId=fReference[0]}
  [1230] = {x=-211, z=176, rx=180, rz=91.364, shoulder=lefty, elbow=epositive, wrist=wpositive, fatherId=fReference[0]}
  [1231] = {x=-211, z=176, rx=180, rz=91.364, shoulder=lefty, elbow=epositive, wrist=wpositive, fatherId=fReference[0]}
  [1232] = {x=-211, z=276, rx=180, rz=91.364, shoulder=lefty, elbow=epositive, wrist=wpositive, fatherId=fReference[0]}
  [1233] = {x=-211, z=298, rx=180, rz=91.364, shoulder=lefty, elbow=epositive, wrist=wpositive, fatherId=fReference[0]}
  [1234] = {x=-211, z=198, rx=180, rz=91.364, shoulder=lefty, elbow=epositive, wrist=wpositive, fatherId=fReference[0]}
  [1235] = {x=-211, z=198, rx=180, rz=91.364, shoulder=lefty, elbow=epositive, wrist=wpositive, fatherId=fReference[0]}
  [1236] = {x=-210.761, y=10.04, z=198, rx=180, rz=94.091, shoulder=lefty, elbow=epositive, wrist=wpositive, fatherId=fReference[0]}
  [1237] = {x=-210.045, y=20.057, z=198, rx=180, rz=96.818, shoulder=lefty, elbow=epositive, wrist=wpositive, fatherId=fReference[0]}
  [1238] = {x=-208.852, y=30.028, z=198, rx=180, rz=99.545, shoulder=lefty, elbow=epositive, wrist=wpositive, fatherId=fReference[0]}
  [1239] = {x=-207.187, y=39.932, z=198, rx=180, rz=102.273, shoulder=lefty, elbow=epositive, wrist=wpositive, fatherId=fReference[0]}
  [1240] = {x=-205.052, y=49.745, z=198, rx=180, rz=105, shoulder=lefty, elbow=epositive, wrist=wpositive, fatherId=fReference[0]}
  [1241] = {x=-202.453, y=59.446, z=198, rx=180, rz=107.727, shoulder=lefty, elbow=epositive, wrist=wpositive, fatherId=fReference[0]}
  [1242] = {x=-199.395, y=69.011, z=198, rx=180, rz=110.455, shoulder=lefty, elbow=epositive, wrist=wpositive, fatherId=fReference[0]}
  [1243] = {x=-195.886, y=78.421, z=198, rx=180, rz=113.182, shoulder=lefty, elbow=epositive, wrist=wpositive, fatherId=fReference[0]}
  [1244] = {x=-191.932, y=87.653, z=198, rx=180, rz=115.909, shoulder=lefty, elbow=epositive, wrist=wpositive, fatherId=fReference[0]}
  [1245] = {x=-187.544, y=96.686, z=198, rx=180, rz=118.636, shoulder=lefty, elbow=epositive, wrist=wpositive, fatherId=fReference[0]}
  [1246] = {x=-182.731, y=105.5, z=198, rx=-180, rz=121.364, shoulder=lefty, elbow=epositive, wrist=wpositive, fatherId=fReference[0]}
  [1247] = {x=-177.505, y=114.075, z=198, rx=180, rz=124.091, shoulder=lefty, elbow=epositive, wrist=wpositive, fatherId=fReference[0]}
  [1248] = {x=-171.876, y=122.392, z=198, rx=180, rz=126.818, shoulder=lefty, elbow=epositive, wrist=wpositive, fatherId=fReference[0]}
  [1249] = {x=-165.857, y=130.432, z=198, rx=-180, rz=129.545, shoulder=lefty, elbow=epositive, wrist=wpositive, fatherId=fReference[0]}
  [1250] = {x=-159.463, y=138.176, z=198, rx=180, rz=132.273, shoulder=lefty, elbow=epositive, wrist=wpositive, fatherId=fReference[0]}
  [1251] = {x=-152.708, y=145.607, z=198, rx=-180, rz=135, shoulder=lefty, elbow=epositive, wrist=wpositive, fatherId=fReference[0]}
  [1252] = {x=-145.607, y=152.708, z=198, rx=-180, rz=137.727, shoulder=lefty, elbow=epositive, wrist=wpositive, fatherId=fReference[0]}
  [1253] = {x=-138.176, y=159.463, z=198, rx=180, rz=140.455, shoulder=lefty, elbow=epositive, wrist=wpositive, fatherId=fReference[0]}
  [1254] = {x=-130.432, y=165.857, z=198, rx=-180, rz=143.182, shoulder=lefty, elbow=epositive, wrist=wpositive, fatherId=fReference[0]}
  [1255] = {x=-122.392, y=171.876, z=198, rx=180, rz=145.909, shoulder=lefty, elbow=epositive, wrist=wpositive, fatherId=fReference[0]}
  [1256] = {x=-114.075, y=177.505, z=198, rx=180, rz=148.636, shoulder=lefty, elbow=epositive, wrist=wpositive, fatherId=fReference[0]}
  [1257] = {x=-105.5, y=182.731, z=198, rx=-180, rz=151.364, shoulder=lefty, elbow=epositive, wrist=wpositive, fatherId=fReference[0]}
  [1258] = {x=-96.686, y=187.544, z=198, rx=-180, rz=154.091, shoulder=lefty, elbow=epositive, wrist=wpositive, fatherId=fReference[0]}
  [1259] = {x=-87.653, y=191.932, z=198, rx=180, rz=156.818, shoulder=lefty, elbow=epositive, wrist=wpositive, fatherId=fReference[0]}
  [1260] = {x=-78.421, y=195.886, z=198, rx=-180, rz=159.545, shoulder=lefty, elbow=epositive, wrist=wpositive, fatherId=fReference[0]}
  [1261] = {x=-69.011, y=199.395, z=198, rx=180, rz=162.273, shoulder=lefty, elbow=epositive, wrist=wpositive, fatherId=fReference[0]}
  [1262] = {x=-59.446, y=202.453, z=198, rx=180, rz=165, shoulder=lefty, elbow=epositive, wrist=wpositive, fatherId=fReference[0]}
  [1263] = {x=-49.745, y=205.052, z=198, rx=180, rz=167.727, shoulder=lefty, elbow=epositive, wrist=wpositive, fatherId=fReference[0]}
  [1264] = {x=-39.932, y=207.187, z=198, rx=-180, rz=170.455, shoulder=lefty, elbow=epositive, wrist=wpositive, fatherId=fReference[0]}
  [1265] = {x=-30.028, y=208.852, z=198, rx=180, rz=173.182, shoulder=lefty, elbow=epositive, wrist=wpositive, fatherId=fReference[0]}
  [1266] = {x=-20.057, y=210.045, z=198, rx=180, rz=175.909, shoulder=lefty, elbow=epositive, wrist=wpositive, fatherId=fReference[0]}
  [1267] = {x=-10.04, y=210.761, z=198, rx=-180, rz=178.636, shoulder=lefty, elbow=epositive, wrist=wpositive, fatherId=fReference[0]}
  [1268] = {y=211, z=198, rx=-180, rz=-178.636, shoulder=lefty, elbow=epositive, wrist=wpositive, fatherId=fReference[0]}
  [1269] = {x=10.04, y=210.761, z=198, rx=-180, rz=-175.909, shoulder=lefty, elbow=epositive, wrist=wpositive, fatherId=fReference[0]}
  [1270] = {x=20.057, y=210.045, z=198, rx=180, rz=-173.182, shoulder=lefty, elbow=epositive, wrist=wpositive, fatherId=fReference[0]}
  [1271] = {x=30.028, y=208.852, z=198, rx=180, rz=-170.455, shoulder=lefty, elbow=epositive, wrist=wpositive, fatherId=fReference[0]}
  [1272] = {x=39.932, y=207.187, z=198, rx=180, rz=-167.727, shoulder=lefty, elbow=epositive, wrist=wpositive, fatherId=fReference[0]}
  [1273] = {x=49.745, y=205.052, z=198, rx=-180, rz=-165, shoulder=lefty, elbow=epositive, wrist=wpositive, fatherId=fReference[0]}
  [1274] = {x=59.446, y=202.453, z=198, rx=-180, rz=-162.273, shoulder=lefty, elbow=epositive, wrist=wpositive, fatherId=fReference[0]}
  [1275] = {x=69.011, y=199.395, z=198, rx=-180, rz=-159.545, shoulder=lefty, elbow=epositive, wrist=wpositive, fatherId=fReference[0]}
  [1276] = {x=78.421, y=195.886, z=198, rx=-180, rz=-156.818, shoulder=lefty, elbow=epositive, wrist=wpositive, fatherId=fReference[0]}
  [1277] = {x=87.653, y=191.932, z=198, rx=-180, rz=-154.091, shoulder=lefty, elbow=epositive, wrist=wpositive, fatherId=fReference[0]}
  [1278] = {x=96.686, y=187.544, z=198, rx=-180, rz=-151.364, shoulder=lefty, elbow=epositive, wrist=wpositive, fatherId=fReference[0]}
  [1279] = {x=105.5, y=182.731, z=198, rx=-180, rz=-148.636, shoulder=lefty, elbow=epositive, wrist=wpositive, fatherId=fReference[0]}
  [1280] = {x=114.075, y=177.505, z=198, rx=180, rz=-145.909, shoulder=lefty, elbow=epositive, wrist=wpositive, fatherId=fReference[0]}
  [1281] = {x=122.392, y=171.876, z=198, rx=180, rz=-143.182, shoulder=lefty, elbow=epositive, wrist=wpositive, fatherId=fReference[0]}
  [1282] = {x=130.432, y=165.857, z=198, rx=-180, rz=-140.455, shoulder=lefty, elbow=epositive, wrist=wpositive, fatherId=fReference[0]}
  [1283] = {x=138.176, y=159.463, z=198, rx=-180, rz=-137.727, shoulder=lefty, elbow=epositive, wrist=wpositive, fatherId=fReference[0]}
  [1284] = {x=145.607, y=152.708, z=198, rx=-180, rz=-135, shoulder=lefty, elbow=epositive, wrist=wpositive, fatherId=fReference[0]}
  [1285] = {x=152.708, y=145.607, z=198, rx=-180, rz=-132.273, shoulder=lefty, elbow=epositive, wrist=wpositive, fatherId=fReference[0]}
  [1286] = {x=159.463, y=138.176, z=198, rx=-180, rz=-129.545, shoulder=lefty, elbow=epositive, wrist=wpositive, fatherId=fReference[0]}
  [1287] = {x=165.857, y=130.432, z=198, rx=-180, rz=-126.818, shoulder=lefty, elbow=epositive, wrist=wpositive, fatherId=fReference[0]}
  [1288] = {x=171.876, y=122.392, z=198, rx=-180, rz=-124.091, shoulder=lefty, elbow=epositive, wrist=wpositive, fatherId=fReference[0]}
  [1289] = {x=177.505, y=114.075, z=198, rx=-180, rz=-121.364, shoulder=lefty, elbow=epositive, wrist=wpositive, fatherId=fReference[0]}
  [1290] = {x=182.731, y=105.5, z=198, rx=-180, rz=-118.636, shoulder=lefty, elbow=epositive, wrist=wpositive, fatherId=fReference[0]}
  [1291] = {x=187.544, y=96.686, z=198, rx=-180, rz=-115.909, shoulder=lefty, elbow=epositive, wrist=wpositive, fatherId=fReference[0]}
  [1292] = {x=191.932, y=87.653, z=198, rx=-180, rz=-113.182, shoulder=lefty, elbow=epositive, wrist=wpositive, fatherId=fReference[0]}
  [1293] = {x=195.886, y=78.421, z=198, rx=-180, rz=-110.455, shoulder=lefty, elbow=epositive, wrist=wpositive, fatherId=fReference[0]}
  [1294] = {x=199.395, y=69.011, z=198, rx=-180, rz=-107.727, shoulder=lefty, elbow=epositive, wrist=wpositive, fatherId=fReference[0]}
  [1295] = {x=202.453, y=59.446, z=198, rx=-180, rz=-105, shoulder=lefty, elbow=epositive, wrist=wpositive, fatherId=fReference[0]}
  [1296] = {x=205.052, y=49.745, z=198, rx=-180, rz=-102.273, shoulder=lefty, elbow=epositive, wrist=wpositive, fatherId=fReference[0]}
  [1297] = {x=207.187, y=39.932, z=198, rx=-180, rz=-99.545, shoulder=lefty, elbow=epositive, wrist=wpositive, fatherId=fReference[0]}
  [1298] = {x=208.852, y=30.028, z=198, rx=-180, rz=-96.818, shoulder=lefty, elbow=epositive, wrist=wpositive, fatherId=fReference[0]}
  [1299] = {x=210.045, y=20.057, z=198, rx=-180, rz=-94.091, shoulder=lefty, elbow=epositive, wrist=wpositive, fatherId=fReference[0]}
  [1300] = {x=210.761, y=10.04, z=198, rx=-180, rz=-91.364, shoulder=lefty, elbow=epositive, wrist=wpositive, fatherId=fReference[0]}
  [1301] = {x=211, z=198, rx=180, rz=-88.636, shoulder=lefty, elbow=epositive, wrist=wpositive, fatherId=fReference[0]}
  [1302] = {x=210.761, y=-10.04, z=198, rx=180, rz=-85.909, shoulder=lefty, elbow=epositive, wrist=wpositive, fatherId=fReference[0]}
  [1303] = {x=210.045, y=-20.057, z=198, rx=180, rz=-83.182, shoulder=lefty, elbow=epositive, wrist=wpositive, fatherId=fReference[0]}
  [1304] = {x=208.852, y=-30.028, z=198, rx=180, rz=-80.455, shoulder=lefty, elbow=epositive, wrist=wpositive, fatherId=fReference[0]}
  [1305] = {x=207.187, y=-39.932, z=198, rx=180, rz=-77.727, shoulder=lefty, elbow=epositive, wrist=wpositive, fatherId=fReference[0]}
  [1306] = {x=205.052, y=-49.745, z=198, rx=180, rz=-75, shoulder=lefty, elbow=epositive, wrist=wpositive, fatherId=fReference[0]}
  [1307] = {x=202.453, y=-59.446, z=198, rx=180, rz=-72.273, shoulder=lefty, elbow=epositive, wrist=wpositive, fatherId=fReference[0]}
  [1308] = {x=199.395, y=-69.011, z=198, rx=-180, rz=-69.545, shoulder=lefty, elbow=epositive, wrist=wpositive, fatherId=fReference[0]}
  [1309] = {x=195.886, y=-78.421, z=198, rx=180, rz=-66.818, shoulder=lefty, elbow=epositive, wrist=wpositive, fatherId=fReference[0]}
  [1310] = {x=191.932, y=-87.653, z=198, rx=180, rz=-64.091, shoulder=lefty, elbow=epositive, wrist=wpositive, fatherId=fReference[0]}
  [1311] = {x=187.544, y=-96.686, z=198, rx=180, rz=-61.364, shoulder=lefty, elbow=epositive, wrist=wpositive, fatherId=fReference[0]}
  [1312] = {x=182.731, y=-105.5, z=198, rx=180, rz=-58.636, shoulder=lefty, elbow=epositive, wrist=wpositive, fatherId=fReference[0]}
  [1313] = {x=177.505, y=-114.075, z=198, rx=180, rz=-55.909, shoulder=lefty, elbow=epositive, wrist=wpositive, fatherId=fReference[0]}
  [1314] = {x=171.876, y=-122.392, z=198, rx=-180, rz=-53.182, shoulder=lefty, elbow=epositive, wrist=wpositive, fatherId=fReference[0]}
  [1315] = {x=165.857, y=-130.432, z=198, rx=180, rz=-50.455, shoulder=lefty, elbow=epositive, wrist=wpositive, fatherId=fReference[0]}
  [1316] = {x=159.463, y=-138.176, z=198, rx=180, rz=-47.727, shoulder=lefty, elbow=epositive, wrist=wpositive, fatherId=fReference[0]}
  [1317] = {x=152.708, y=-145.607, z=198, rx=180, rz=-45, shoulder=lefty, elbow=epositive, wrist=wpositive, fatherId=fReference[0]}
  [1318] = {x=145.607, y=-152.708, z=198, rx=180, rz=-42.273, shoulder=lefty, elbow=epositive, wrist=wpositive, fatherId=fReference[0]}
  [1319] = {x=138.176, y=-159.463, z=198, rx=180, rz=-39.545, shoulder=lefty, elbow=epositive, wrist=wpositive, fatherId=fReference[0]}
  [1320] = {x=130.432, y=-165.857, z=198, rx=180, rz=-36.818, shoulder=lefty, elbow=epositive, wrist=wpositive, fatherId=fReference[0]}
  [1321] = {x=122.392, y=-171.876, z=198, rx=-180, rz=-34.091, shoulder=lefty, elbow=epositive, wrist=wpositive, fatherId=fReference[0]}
  [1322] = {x=114.075, y=-177.505, z=198, rx=-180, rz=-31.364, shoulder=lefty, elbow=epositive, wrist=wpositive, fatherId=fReference[0]}
  [1323] = {x=105.5, y=-182.731, z=198, rx=180, rz=-28.636, shoulder=lefty, elbow=epositive, wrist=wpositive, fatherId=fReference[0]}
  [1324] = {x=96.686, y=-187.544, z=198, rx=-180, rz=-25.909, shoulder=lefty, elbow=epositive, wrist=wpositive, fatherId=fReference[0]}
  [1325] = {x=87.653, y=-191.932, z=198, rx=-180, rz=-23.182, shoulder=lefty, elbow=epositive, wrist=wpositive, fatherId=fReference[0]}
  [1326] = {x=78.421, y=-195.886, z=198, rx=180, rz=-20.455, shoulder=lefty, elbow=epositive, wrist=wpositive, fatherId=fReference[0]}
  [1327] = {x=69.011, y=-199.395, z=198, rx=180, rz=-17.727, shoulder=lefty, elbow=epositive, wrist=wpositive, fatherId=fReference[0]}
  [1328] = {x=59.446, y=-202.453, z=198, rx=-180, rz=-15, shoulder=lefty, elbow=epositive, wrist=wpositive, fatherId=fReference[0]}
  [1329] = {x=49.745, y=-205.052, z=198, rx=-180, rz=-12.273, shoulder=lefty, elbow=epositive, wrist=wpositive, fatherId=fReference[0]}
  [1330] = {x=39.932, y=-207.187, z=198, rx=-180, rz=-9.545, shoulder=lefty, elbow=epositive, wrist=wpositive, fatherId=fReference[0]}
  [1331] = {x=30.028, y=-208.852, z=198, rx=180, rz=-6.818, shoulder=lefty, elbow=epositive, wrist=wpositive, fatherId=fReference[0]}
  [1332] = {x=20.057, y=-210.045, z=198, rx=180, rz=-4.091, shoulder=lefty, elbow=epositive, wrist=wpositive, fatherId=fReference[0]}
  [1333] = {x=10.04, y=-210.761, z=198, rx=180, rz=-1.364, shoulder=lefty, elbow=epositive, wrist=wpositive, fatherId=fReference[0]}
  [1334] = {y=-211, z=198, rx=180, rz=1.364, shoulder=lefty, elbow=epositive, wrist=wpositive, fatherId=fReference[0]}
  [1335] = {x=-10.04, y=-210.761, z=198, rx=180, rz=4.091, shoulder=lefty, elbow=epositive, wrist=wpositive, fatherId=fReference[0]}
  [1336] = {x=-20.057, y=-210.045, z=198, rx=-180, rz=6.818, shoulder=lefty, elbow=epositive, wrist=wpositive, fatherId=fReference[0]}
  [1337] = {x=-30.028, y=-208.852, z=198, rx=-180, rz=9.545, shoulder=lefty, elbow=epositive, wrist=wpositive, fatherId=fReference[0]}
  [1338] = {x=-39.932, y=-207.187, z=198, rx=-180, rz=12.273, shoulder=lefty, elbow=epositive, wrist=wpositive, fatherId=fReference[0]}
  [1339] = {x=-49.745, y=-205.052, z=198, rx=-180, rz=15, shoulder=lefty, elbow=epositive, wrist=wpositive, fatherId=fReference[0]}
  [1340] = {x=-59.446, y=-202.453, z=198, rx=180, rz=17.727, shoulder=lefty, elbow=epositive, wrist=wpositive, fatherId=fReference[0]}
  [1341] = {x=-69.011, y=-199.395, z=198, rx=-180, rz=20.455, shoulder=lefty, elbow=epositive, wrist=wpositive, fatherId=fReference[0]}
  [1342] = {x=-78.421, y=-195.886, z=198, rx=-180, rz=23.182, shoulder=lefty, elbow=epositive, wrist=wpositive, fatherId=fReference[0]}
  [1343] = {x=-87.653, y=-191.932, z=198, rx=-180, rz=25.909, shoulder=lefty, elbow=epositive, wrist=wpositive, fatherId=fReference[0]}
  [1344] = {x=-96.686, y=-187.544, z=198, rx=-180, rz=28.636, shoulder=lefty, elbow=epositive, wrist=wpositive, fatherId=fReference[0]}
  [1345] = {x=-105.5, y=-182.731, z=198, rx=180, rz=31.364, shoulder=lefty, elbow=epositive, wrist=wpositive, fatherId=fReference[0]}
  [1346] = {x=-114.075, y=-177.505, z=198, rx=180, rz=34.091, shoulder=lefty, elbow=epositive, wrist=wpositive, fatherId=fReference[0]}
  [1347] = {x=-122.392, y=-171.876, z=198, rx=-180, rz=36.818, shoulder=lefty, elbow=epositive, wrist=wpositive, fatherId=fReference[0]}
  [1348] = {x=-130.432, y=-165.857, z=198, rx=-180, rz=39.545, shoulder=lefty, elbow=epositive, wrist=wpositive, fatherId=fReference[0]}
  [1349] = {x=-138.176, y=-159.463, z=198, rx=-180, rz=42.273, shoulder=lefty, elbow=epositive, wrist=wpositive, fatherId=fReference[0]}
  [1350] = {x=-145.607, y=-152.708, z=198, rx=180, rz=45, shoulder=lefty, elbow=epositive, wrist=wpositive, fatherId=fReference[0]}
  [1351] = {x=-152.708, y=-145.607, z=198, rx=-180, rz=47.727, shoulder=lefty, elbow=epositive, wrist=wpositive, fatherId=fReference[0]}
  [1352] = {x=-159.463, y=-138.176, z=198, rx=-180, rz=50.455, shoulder=lefty, elbow=epositive, wrist=wpositive, fatherId=fReference[0]}
  [1353] = {x=-165.857, y=-130.432, z=198, rx=-180, rz=53.182, shoulder=lefty, elbow=epositive, wrist=wpositive, fatherId=fReference[0]}
  [1354] = {x=-171.876, y=-122.392, z=198, rx=-180, rz=55.909, shoulder=lefty, elbow=epositive, wrist=wpositive, fatherId=fReference[0]}
  [1355] = {x=-177.505, y=-114.075, z=198, rx=-180, rz=58.636, shoulder=lefty, elbow=epositive, wrist=wpositive, fatherId=fReference[0]}
  [1356] = {x=-182.731, y=-105.5, z=198, rx=-180, rz=61.364, shoulder=lefty, elbow=epositive, wrist=wpositive, fatherId=fReference[0]}
  [1357] = {x=-187.544, y=-96.686, z=198, rx=-180, rz=64.091, shoulder=lefty, elbow=epositive, wrist=wpositive, fatherId=fReference[0]}
  [1358] = {x=-191.932, y=-87.653, z=198, rx=-180, rz=66.818, shoulder=lefty, elbow=epositive, wrist=wpositive, fatherId=fReference[0]}
  [1359] = {x=-195.886, y=-78.421, z=198, rx=-180, rz=69.545, shoulder=lefty, elbow=epositive, wrist=wpositive, fatherId=fReference[0]}
  [1360] = {x=-199.395, y=-69.011, z=198, rx=-180, rz=72.273, shoulder=lefty, elbow=epositive, wrist=wpositive, fatherId=fReference[0]}
  [1361] = {x=-202.453, y=-59.446, z=198, rx=-180, rz=75, shoulder=lefty, elbow=epositive, wrist=wpositive, fatherId=fReference[0]}
  [1362] = {x=-205.052, y=-49.745, z=198, rx=-180, rz=77.727, shoulder=lefty, elbow=epositive, wrist=wpositive, fatherId=fReference[0]}
  [1363] = {x=-207.187, y=-39.932, z=198, rx=-180, rz=80.455, shoulder=lefty, elbow=epositive, wrist=wpositive, fatherId=fReference[0]}
  [1364] = {x=-208.852, y=-30.028, z=198, rx=-180, rz=83.182, shoulder=lefty, elbow=epositive, wrist=wpositive, fatherId=fReference[0]}
  [1365] = {x=-210.045, y=-20.057, z=198, rx=-180, rz=85.909, shoulder=lefty, elbow=epositive, wrist=wpositive, fatherId=fReference[0]}
  [1366] = {x=-210.761, y=-10.04, z=198, rx=-180, rz=88.636, shoulder=lefty, elbow=epositive, wrist=wpositive, fatherId=fReference[0]}
  [1367] = {x=-211, z=198, rx=-180, rz=88.636, shoulder=lefty, elbow=epositive, wrist=wpositive, fatherId=fReference[0]}
  [1368] = {x=-211, z=198, rx=-180, rz=88.636, shoulder=lefty, elbow=epositive, wrist=wpositive, fatherId=fReference[0]}
  [1369] = {x=-211, z=298, rx=-180, rz=88.636, shoulder=lefty, elbow=epositive, wrist=wpositive, fatherId=fReference[0]}
public tool tTool = {z=452, fatherId=flange[0], ioLink=valve1}
dio doValve1 = {link=valve1}
aio Tpompe = {link=CanIO\RemIO\remio0_QW}
